(* CoDeSys 2.3.9.40 project: Атмосфера 02.12.15.pro *)
(* Libraries: Util.lib 18.5.10 14:14:28, STANDARD.LIB 4.10.05 10:14:46, IECSFC.LIB 13.4.06 14:51:28, ANALYZATION.LIB 5.10.99 08:05:06 *)

(* PLC configuration (modules and I/O channels)
Fast discrete inputs [I_SIMPLE_INPUT] node 0, in %IB0 out %QB0 {Filtrationtime = 10}
  AT %IX0.0 [BitInput] PUSK_SYS
  AT %IX0.1 [BitInput] STOP_SYS
  AT %IX0.2 [BitInput] gribok
  AT %IX0.3 [BitInput] avto_all
Discrete inputs [ID130] node 1, in %IB1 out %QB1 {Filtrationtime_GeneralINP = 10; Visibility = No; PinCount = 32}
  AT %IB1.0 [ByteInput] 8 discrete inputs
  AT %IB1.1 [ByteInput] 8 discrete inputs
  AT %IB1.2 [ByteInput] 8 discrete inputs
  AT %IB1.3 [ByteInput] 8 discrete inputs
Fast discrete outputs [OWEN_ID570] node 2, in %IB2 out %QB2 {SafeValueBool = FALSE; SafeValueBool = FALSE; SafeValueBool = FALSE; SafeValueBool = FALSE; Visibility = No}
  AT %QX2.0 [BitOutput] ready_LK3
  AT %QX2.1 [BitOutput] avaria
  AT %QX2.2 [BitOutput] metall
  AT %QX2.3 [BitOutput] ready_LK10
Discrete outputs [ID131] node 3, in %IB3 out %QB3 {SafeValueByte = 0; SafeValueByte = 0; SafeValueByteM = 0; Visibility = No; PinCount = 24}
  AT %QB3.0 [ByteOutput] 8 discrete outputs
  AT %QB3.1 [ByteOutput] 8 discrete outputs
  AT %QB3.2 [ByteOutput] 4 discrete outputs
Special input [ID103] node 4, in %IB4 out %QB4 {Filtrationtime = 1000; PinCount = 1; WatchDogPeriod = 400; PollPeriod = 3000; Visibility = No}
  AT %IX4.0 [BitInput] Special input
Special output [ID104] node 5, in %IB5 out %QB5 {Visibility = No; PinCount = 1}
  AT %QX5.0 [BitOutput] Special output
Button [ID003] node 6, in %IB6 out %QB6
  AT %IX6.0 [BitInput] Button Start/Stop
ModBus (Master) [MODBUS_MASTER_ID450] node 7, in %IB7 out %QB7 {Visibility = No}
  AT %QD7.0 [DWordOutput] Last address
  AT %QW7.1 [WordOutput] Last error
  RS-485-2 [COM3_USART] node 0, in %IB7.0 out %QB7.0 {CommunicationSpeed = 38400; Parity = NO PARITY CHECK; BitLength = 8 bits; StopLength = One stop bit; InterfaceType = RS485; FrameOriented = RTU; Timeout = 0; Visibility = No}
  Universal Modbus device [ID2000] node 1, in %IB7.1 out %QB7.1 {ModuleIP = 10:0:0:223; ServiceTimeout = 150; TCPport = 502; NetMode = Serial; ModuleSlaveAddress = 10; RequestType = By poll time; PeriodOfService = 100; Visibility = No; RepeatCounter = 0; ByteSequence = Trace_mode}
    AT %QB7.1.0 [ComChannel] LK10
AT %IB7.1.0.0 [ByteInput]
AT %QW7.1.1.0 [WordOutput] KM1_LK10
AT %IW7.1.2.0 [WordInput]
Universal Modbus device [ID2000] node 2, in %IB7.2 out %QB7.2 {ModuleIP = 10:0:0:223; ServiceTimeout = 150; TCPport = 502; NetMode = Serial; ModuleSlaveAddress = 11; RequestType = By poll time; PeriodOfService = 100; Visibility = No; RepeatCounter = 0; ByteSequence = Trace_mode}
  AT %QB7.2.0 [ComChannel] LK11
AT %IB7.2.0.0 [ByteInput]
AT %QW7.2.1.0 [WordOutput] KM1_LK11
AT %IW7.2.2.0 [WordInput]
Universal Modbus device [ID2000] node 3, in %IB7.3 out %QB7.3 {ModuleIP = 10:0:0:223; ServiceTimeout = 150; TCPport = 502; NetMode = Serial; ModuleSlaveAddress = 12; RequestType = By poll time; PeriodOfService = 100; Visibility = No; RepeatCounter = 0; ByteSequence = Trace_mode}
  AT %QB7.3.0 [ComChannel] LK12
AT %IB7.3.0.0 [ByteInput]
AT %QW7.3.1.0 [WordOutput] KM1_LK12
AT %IW7.3.2.0 [WordInput]
Universal Modbus device [ID2000] node 4, in %IB7.4 out %QB7.4 {ModuleIP = 10:0:0:223; ServiceTimeout = 150; TCPport = 502; NetMode = Serial; ModuleSlaveAddress = 13; RequestType = By poll time; PeriodOfService = 100; Visibility = No; RepeatCounter = 0; ByteSequence = Trace_mode}
  AT %QB7.4.0 [ComChannel] LK13
AT %IB7.4.0.0 [ByteInput]
AT %QW7.4.1.0 [WordOutput] KM1_LK13
AT %IW7.4.2.0 [WordInput]
Universal Modbus device [ID2000] node 5, in %IB7.5 out %QB7.5 {ModuleIP = 10:0:0:223; ServiceTimeout = 150; TCPport = 502; NetMode = Serial; ModuleSlaveAddress = 14; RequestType = By poll time; PeriodOfService = 100; Visibility = No; RepeatCounter = 0; ByteSequence = Trace_mode}
  AT %QB7.5.0 [ComChannel] GR3
AT %IB7.5.0.0 [ByteInput]
AT %QW7.5.1.0 [WordOutput] KM1_GR3
Universal Modbus device [ID2000] node 6, in %IB7.6 out %QB7.6 {ModuleIP = 10:0:0:223; ServiceTimeout = 150; TCPport = 502; NetMode = Serial; ModuleSlaveAddress = 6; RequestType = By poll time; PeriodOfService = 100; Visibility = No; RepeatCounter = 0; ByteSequence = Trace_mode}
  AT %QB7.6.0 [ComChannel] LK6
AT %IB7.6.0.0 [ByteInput]
AT %QW7.6.1.0 [WordOutput] KM1_LK6
AT %IW7.6.2.0 [WordInput]
Universal Modbus device [ID2000] node 7, in %IB7.7 out %QB7.7 {ModuleIP = 10:0:0:223; ServiceTimeout = 150; TCPport = 502; NetMode = Serial; ModuleSlaveAddress = 9; RequestType = By poll time; PeriodOfService = 100; Visibility = No; RepeatCounter = 0; ByteSequence = Trace_mode}
  AT %QB7.7.0 [ComChannel] LK9
AT %IB7.7.0.0 [ByteInput]
AT %QW7.7.1.0 [WordOutput] KM1_LK9
AT %IW7.7.2.0 [WordInput]
Universal Modbus device [ID2000] node 8, in %IB7.8 out %QB7.8 {ModuleIP = 10:0:0:223; ServiceTimeout = 150; TCPport = 502; NetMode = Serial; ModuleSlaveAddress = 18; RequestType = By poll time; PeriodOfService = 100; Visibility = No; RepeatCounter = 0; ByteSequence = Trace_mode}
  AT %QB7.8.0 [ComChannel] LP1_3 mod1
AT %IB7.8.0.0 [ByteInput]
AT %QW7.8.1.0 [WordOutput] KM1_LP1_3
Universal Modbus device [ID2000] node 9, in %IB7.9 out %QB7.9 {ModuleIP = 10:0:0:223; ServiceTimeout = 150; TCPport = 502; NetMode = Serial; ModuleSlaveAddress = 19; RequestType = By poll time; PeriodOfService = 100; Visibility = No; RepeatCounter = 0; ByteSequence = Trace_mode}
  AT %QB7.9.0 [ComChannel] LP1_3 mod2
AT %IB7.9.0.0 [ByteInput]
AT %QW7.9.1.0 [WordOutput] KM2345_LP1_3_byte
AT %IW7.9.2.0 [WordInput]
AT %IW7.9.3.0 [WordInput]
AT %IW7.9.4.0 [WordInput]
Universal Modbus device [ID2000] node 10, in %IB7.10 out %QB7.10 {ModuleIP = 10:0:0:223; ServiceTimeout = 150; TCPport = 502; NetMode = Serial; ModuleSlaveAddress = 15; RequestType = By poll time; PeriodOfService = 100; Visibility = No; RepeatCounter = 0; ByteSequence = Trace_mode}
  AT %QB7.10.0 [ComChannel] GR2
AT %IB7.10.0.0 [ByteInput]
AT %QW7.10.1.0 [WordOutput] KM1_GR2
Universal Modbus device [ID2000] node 11, in %IB7.11 out %QB7.11 {ModuleIP = 10:0:0:223; ServiceTimeout = 150; TCPport = 502; NetMode = Serial; ModuleSlaveAddress = 4; RequestType = By poll time; PeriodOfService = 100; Visibility = No; RepeatCounter = 0; ByteSequence = Trace_mode}
  AT %QB7.11.0 [ComChannel] LK4
AT %IB7.11.0.0 [ByteInput]
AT %QW7.11.1.0 [WordOutput] KM1_LK4
AT %IW7.11.2.0 [WordInput]
Universal Modbus device [ID2000] node 12, in %IB7.12 out %QB7.12 {ModuleIP = 10:0:0:223; ServiceTimeout = 150; TCPport = 502; NetMode = Serial; ModuleSlaveAddress = 1; RequestType = By poll time; PeriodOfService = 100; Visibility = No; RepeatCounter = 0; ByteSequence = Trace_mode}
  AT %QB7.12.0 [ComChannel] GR1
AT %IB7.12.0.0 [ByteInput]
AT %QW7.12.1.0 [WordOutput] KM1_GR1
Universal Modbus device [ID2000] node 13, in %IB7.13 out %QB7.13 {ModuleIP = 10:0:0:223; ServiceTimeout = 150; TCPport = 502; NetMode = Serial; ModuleSlaveAddress = 2; RequestType = By poll time; PeriodOfService = 100; Visibility = No; RepeatCounter = 0; ByteSequence = Trace_mode}
  AT %QB7.13.0 [ComChannel] LK2
AT %IB7.13.0.0 [ByteInput]
AT %QW7.13.1.0 [WordOutput] KM1_LK2
AT %IW7.13.2.0 [WordInput]
Universal Modbus device [ID2000] node 14, in %IB7.14 out %QB7.14 {ModuleIP = 10:0:0:223; ServiceTimeout = 150; TCPport = 502; NetMode = Serial; ModuleSlaveAddress = 3; RequestType = By poll time; PeriodOfService = 100; Visibility = No; RepeatCounter = 0; ByteSequence = Trace_mode}
  AT %QB7.14.0 [ComChannel] LK3
AT %IB7.14.0.0 [ByteInput]
AT %QW7.14.1.0 [WordOutput] KM1_LK3
AT %IW7.14.2.0 [WordInput]
Universal Modbus device [ID2000] node 15, in %IB7.15 out %QB7.15 {ModuleIP = 10:0:0:223; ServiceTimeout = 150; TCPport = 502; NetMode = Serial; ModuleSlaveAddress = 20; RequestType = By poll time; PeriodOfService = 100; Visibility = No; RepeatCounter = 0; ByteSequence = Trace_mode}
  AT %QB7.15.0 [ComChannel] VP1
AT %IB7.15.0.0 [ByteInput]
AT %QW7.15.1.0 [WordOutput]
Universal Modbus device [ID2000] node 16, in %IB7.16 out %QB7.16 {ModuleIP = 10:0:0:223; ServiceTimeout = 150; TCPport = 502; NetMode = Serial; ModuleSlaveAddress = 27; RequestType = By poll time; PeriodOfService = 100; Visibility = No; RepeatCounter = 0; ByteSequence = Trace_mode}
  AT %QB7.16.0 [ComChannel] Command (0xff - Start)
AT %IB7.16.0.0 [ByteInput]
AT %QW7.16.1.0 [WordOutput] km_byte_cyc
Universal Modbus device [ID2000] node 17, in %IB7.17 out %QB7.17 {ModuleIP = 10:0:0:223; ServiceTimeout = 150; TCPport = 502; NetMode = Serial; ModuleSlaveAddress = 26; RequestType = By poll time; PeriodOfService = 100; Visibility = No; RepeatCounter = 0; ByteSequence = Trace_mode}
  AT %QB7.17.0 [ComChannel] Command (0xff - Start)
AT %QW7.17.0.0 [WordOutput]
AT %QW7.17.1.0 [WordOutput]
AT %QW7.17.2.0 [WordOutput]
AT %QW7.17.3.0 [WordOutput]
AT %QW7.17.4.0 [WordOutput]
AT %QW7.17.5.0 [WordOutput]
AT %QW7.17.6.0 [WordOutput]
AT %QW7.17.7.0 [WordOutput]
Universal Modbus device [ID2000] node 18, in %IB7.18 out %QB7.18 {ModuleIP = 10:0:0:223; ServiceTimeout = 150; TCPport = 502; NetMode = Serial; ModuleSlaveAddress = 44; RequestType = By poll time; PeriodOfService = 100; Visibility = No; RepeatCounter = 0; ByteSequence = Trace_mode}
  AT %QB7.18.0 [ComChannel] Command (0xff - Start)
AT %ID7.18.0.0 [FloatInput]
AT %ID7.18.1.0 [FloatInput]
ModBus (slave) [MODBUS_ID400] node 8, in %IB8 out %QB8 {SlaveIdentificator = 1; Visibility = No}
  Modbus [MODBUS_ID302] node 0, in %IB8.0 out %QB8.0
    TCP [TCP_ID221] node 0, in %IB8.0.0 out %QB8.0.0 {RemotePort = 502; Visibility = No}
  8 bits [8Bit] node 1, in %IB8.1 out %QB8.1
    AT %QB8.1.0 [ByteOutput]
  8 bits [8Bit] node 2, in %IB8.2 out %QB8.2
    AT %QB8.2.0 [ByteOutput]
  8 bits [8Bit] node 3, in %IB8.3 out %QB8.3
    AT %QB8.3.0 [ByteOutput]
  8 bits [8Bit] node 4, in %IB8.4 out %QB8.4
    AT %QB8.4.0 [ByteOutput]
  8 bits [8Bit] node 5, in %IB8.5 out %QB8.5
    AT %QB8.5.0 [ByteOutput]
  8 bits [8Bit] node 6, in %IB8.6 out %QB8.6
    AT %QB8.6.0 [ByteOutput]
  8 bits [8Bit] node 7, in %IB8.7 out %QB8.7
    AT %QB8.7.0 [ByteOutput]
  8 bits [8Bit] node 8, in %IB8.8 out %QB8.8
    AT %QB8.8.0 [ByteOutput]
  8 bits [8Bit] node 9, in %IB8.9 out %QB8.9
    AT %QB8.9.0 [ByteOutput]
  8 bits [8Bit] node 10, in %IB8.10 out %QB8.10
    AT %QB8.10.0 [ByteOutput]
  8 bits [8Bit] node 11, in %IB8.11 out %QB8.11
    AT %QB8.11.0 [ByteOutput]
  8 bits [8Bit] node 12, in %IB8.12 out %QB8.12
    AT %QB8.12.0 [ByteOutput]
  8 bits [8Bit] node 13, in %IB8.13 out %QB8.13
    AT %QB8.13.0 [ByteOutput]
  8 bits [8Bit] node 14, in %IB8.14 out %QB8.14
    AT %QB8.14.0 [ByteOutput]
  8 bits [8Bit] node 15, in %IB8.15 out %QB8.15
    AT %QB8.15.0 [ByteOutput]
  8 bits [8Bit] node 16, in %IB8.16 out %QB8.16
    AT %QB8.16.0 [ByteOutput]
  8 bits [8Bit] node 17, in %IB8.17 out %QB8.17
    AT %QB8.17.0 [ByteOutput]
  8 bits [8Bit] node 18, in %IB8.18 out %QB8.18
    AT %QB8.18.0 [ByteOutput]
  8 bits [8Bit] node 19, in %IB8.19 out %QB8.19
    AT %QB8.19.0 [ByteOutput]
  8 bits [8Bit] node 20, in %IB8.20 out %QB8.20
    AT %QB8.20.0 [ByteOutput]
  8 bits [8Bit] node 21, in %IB8.21 out %QB8.21
    AT %QB8.21.0 [ByteOutput]
  8 bits [8Bit] node 22, in %IB8.22 out %QB8.22
    AT %QB8.22.0 [ByteOutput]
  8 bits [8Bit] node 23, in %IB8.23 out %QB8.23
    AT %QB8.23.0 [ByteOutput]
  8 bits [8Bit] node 24, in %IB8.24 out %QB8.24
    AT %QB8.24.0 [ByteOutput]
  8 bits [8Bit] node 25, in %IB8.25 out %QB8.25
    AT %QB8.25.0 [ByteOutput]
  8 bits [8Bit] node 26, in %IB8.26 out %QB8.26
    AT %QB8.26.0 [ByteOutput]
  8 bits [8Bit] node 27, in %IB8.27 out %QB8.27
    AT %QB8.27.0 [ByteOutput]
  8 bits [8Bit] node 28, in %IB8.28 out %QB8.28
    AT %QB8.28.0 [ByteOutput]
  8 bits [8Bit] node 29, in %IB8.29 out %QB8.29
    AT %QB8.29.0 [ByteOutput]
  8 bits [8Bit] node 30, in %IB8.30 out %QB8.30
    AT %QB8.30.0 [ByteOutput]
  8 bits [8Bit] node 31, in %IB8.31 out %QB8.31
    AT %QB8.31.0 [ByteOutput]
  2 byte [Register] node 32, in %IB8.32 out %QB8.32
    AT %QW8.32.0 [WordOutput] input_Hz_LP4
  2 byte [Register] node 33, in %IB8.33 out %QB8.33
    AT %QW8.33.0 [WordOutput] input_Hz_LP5
  2 byte [Register] node 34, in %IB8.34 out %QB8.34
    AT %QW8.34.0 [WordOutput] LV_GR1_out
  2 byte [Register] node 35, in %IB8.35 out %QB8.35
    AT %QW8.35.0 [WordOutput] LV_LK7_out
  2 byte [Register] node 36, in %IB8.36 out %QB8.36
    AT %QW8.36.0 [WordOutput] LV_LK8_out
  2 byte [Register] node 37, in %IB8.37 out %QB8.37
    AT %QW8.37.0 [WordOutput] output_Hz_LP4_out
  2 byte [Register] node 38, in %IB8.38 out %QB8.38
    AT %QW8.38.0 [WordOutput] output_Hz_LP5_out
  2 byte [Register] node 39, in %IB8.39 out %QB8.39
    AT %QW8.39.0 [WordOutput] LV_D2_out
  Float [Float] node 40, in %IB8.40 out %QB8.40
    AT %QD8.40.0 [FloatOutput] ust_LV2_GR1
  Float [Float] node 41, in %IB8.41 out %QB8.41
    AT %QD8.41.0 [FloatOutput] ust_LV1_GR1
  Float [Float] node 42, in %IB8.42 out %QB8.42
    AT %QD8.42.0 [FloatOutput] ust_LV2_LK7
  Float [Float] node 43, in %IB8.43 out %QB8.43
    AT %QD8.43.0 [FloatOutput] ust_LV1_LK7
  Float [Float] node 44, in %IB8.44 out %QB8.44
    AT %QD8.44.0 [FloatOutput] ust_LV1_LK7
  Float [Float] node 45, in %IB8.45 out %QB8.45
    AT %QD8.45.0 [FloatOutput] ust_LV1_LK7
  Float [Float] node 46, in %IB8.46 out %QB8.46
    AT %QD8.46.0 [FloatOutput] ust_LV1_LK7
  Float [Float] node 47, in %IB8.47 out %QB8.47
    AT %QD8.47.0 [FloatOutput] ust_LV1_LK7
  2 byte [Register] node 48, in %IB8.48 out %QB8.48
    AT %QW8.48.0 [WordOutput] pusk_LAN_LP4
  2 byte [Register] node 49, in %IB8.49 out %QB8.49
    AT %QW8.49.0 [WordOutput] stop_LAN_LP4
  2 byte [Register] node 50, in %IB8.50 out %QB8.50
    AT %QW8.50.0 [WordOutput] pusk_LAN_LP5
  2 byte [Register] node 51, in %IB8.51 out %QB8.51
    AT %QW8.51.0 [WordOutput] stop_LAN_LP5
  2 byte [Register] node 52, in %IB8.52 out %QB8.52
    AT %QW8.52.0 [WordOutput] pusk_LAN_VP1
  2 byte [Register] node 53, in %IB8.53 out %QB8.53
    AT %QW8.53.0 [WordOutput] stop_LAN_VP1
  2 byte [Register] node 54, in %IB8.54 out %QB8.54
    AT %QW8.54.0 [WordOutput] pusk_lan_LK10
  2 byte [Register] node 55, in %IB8.55 out %QB8.55
    AT %QW8.55.0 [WordOutput] pusk_lan_LK11
  2 byte [Register] node 56, in %IB8.56 out %QB8.56
    AT %QW8.56.0 [WordOutput] pusk_lan_LK12
  2 byte [Register] node 57, in %IB8.57 out %QB8.57
    AT %QW8.57.0 [WordOutput] pusk_lan_LK13
  2 byte [Register] node 58, in %IB8.58 out %QB8.58
    AT %QW8.58.0 [WordOutput] pusk_lan_GR3
  2 byte [Register] node 59, in %IB8.59 out %QB8.59
    AT %QW8.59.0 [WordOutput] pusk_lan_LK7
  2 byte [Register] node 60, in %IB8.60 out %QB8.60
    AT %QW8.60.0 [WordOutput] pusk_lan_LK8
  2 byte [Register] node 61, in %IB8.61 out %QB8.61
    AT %QW8.61.0 [WordOutput] pusk_lan_LK6
  2 byte [Register] node 62, in %IB8.62 out %QB8.62
    AT %QW8.62.0 [WordOutput] pusk_lan_LK9
  2 byte [Register] node 63, in %IB8.63 out %QB8.63
    AT %QW8.63.0 [WordOutput] pusk_lan_LP1_3
  2 byte [Register] node 64, in %IB8.64 out %QB8.64
    AT %QW8.64.0 [WordOutput] pusk_lan_GR2
  2 byte [Register] node 65, in %IB8.65 out %QB8.65
    AT %QW8.65.0 [WordOutput] pusk_lan_LK5
  2 byte [Register] node 66, in %IB8.66 out %QB8.66
    AT %QW8.66.0 [WordOutput] pusk_lan_LK4
  2 byte [Register] node 67, in %IB8.67 out %QB8.67
    AT %QW8.67.0 [WordOutput] pusk_lan_LK3
  2 byte [Register] node 68, in %IB8.68 out %QB8.68
    AT %QW8.68.0 [WordOutput] pusk_lan_GR1
  2 byte [Register] node 69, in %IB8.69 out %QB8.69
    AT %QW8.69.0 [WordOutput] pusk_lan_LK2
  2 byte [Register] node 70, in %IB8.70 out %QB8.70
    AT %QW8.70.0 [WordOutput] stop_lan_LK10
  2 byte [Register] node 71, in %IB8.71 out %QB8.71
    AT %QW8.71.0 [WordOutput] stop_lan_LK11
  2 byte [Register] node 72, in %IB8.72 out %QB8.72
    AT %QW8.72.0 [WordOutput] stop_lan_LK12
  2 byte [Register] node 73, in %IB8.73 out %QB8.73
    AT %QW8.73.0 [WordOutput] stop_lan_LK13
  2 byte [Register] node 74, in %IB8.74 out %QB8.74
    AT %QW8.74.0 [WordOutput] stop_lan_GR3
  2 byte [Register] node 75, in %IB8.75 out %QB8.75
    AT %QW8.75.0 [WordOutput] stop_lan_LK7
  2 byte [Register] node 76, in %IB8.76 out %QB8.76
    AT %QW8.76.0 [WordOutput] stop_lan_LK8
  2 byte [Register] node 77, in %IB8.77 out %QB8.77
    AT %QW8.77.0 [WordOutput] stop_lan_LK6
  2 byte [Register] node 78, in %IB8.78 out %QB8.78
    AT %QW8.78.0 [WordOutput] stop_lan_LK9
  2 byte [Register] node 79, in %IB8.79 out %QB8.79
    AT %QW8.79.0 [WordOutput] stop_lan_LP1_3
  2 byte [Register] node 80, in %IB8.80 out %QB8.80
    AT %QW8.80.0 [WordOutput] stop_lan_GR2
  2 byte [Register] node 81, in %IB8.81 out %QB8.81
    AT %QW8.81.0 [WordOutput] stop_lan_LK5
  2 byte [Register] node 82, in %IB8.82 out %QB8.82
    AT %QW8.82.0 [WordOutput] stop_lan_LK4
  2 byte [Register] node 83, in %IB8.83 out %QB8.83
    AT %QW8.83.0 [WordOutput] stop_lan_LK3
  2 byte [Register] node 84, in %IB8.84 out %QB8.84
    AT %QW8.84.0 [WordOutput] stop_lan_GR1
  2 byte [Register] node 85, in %IB8.85 out %QB8.85
    AT %QW8.85.0 [WordOutput] stop_lan_LK2
  2 byte [Register] node 86, in %IB8.86 out %QB8.86
    AT %QW8.86.0 [WordOutput] stop_LAN_D3
  2 byte [Register] node 87, in %IB8.87 out %QB8.87
    AT %QW8.87.0 [WordOutput] stop_LAN_D4
  2 byte [Register] node 88, in %IB8.88 out %QB8.88
    AT %QW8.88.0 [WordOutput] stop_LAN_D2
  2 byte [Register] node 89, in %IB8.89 out %QB8.89
    AT %QW8.89.0 [WordOutput] pusk_LAN_D2
  2 byte [Register] node 90, in %IB8.90 out %QB8.90
    AT %QW8.90.0 [WordOutput] pusk_LAN_D3
  2 byte [Register] node 91, in %IB8.91 out %QB8.91
    AT %QW8.91.0 [WordOutput] pusk_LAN_D4
  2 byte [Register] node 92, in %IB8.92 out %QB8.92
    AT %QW8.92.0 [WordOutput] pusk_lan_cyclone
  2 byte [Register] node 93, in %IB8.93 out %QB8.93
    AT %QW8.93.0 [WordOutput] stop_lan_cyclone
  Float [Float] node 94, in %IB8.94 out %QB8.94
    AT %QD8.94.0 [FloatOutput] skvaj_in
  Float [Float] node 95, in %IB8.95 out %QB8.95
    AT %QD8.95.0 [FloatOutput] skvaj1_in
  Float [Float] node 96, in %IB8.96 out %QB8.96
    AT %QD8.96.0 [FloatOutput] skvaj2_in
  Float [Float] node 97, in %IB8.97 out %QB8.97
    AT %QD8.97.0 [FloatOutput] skvaj3_in
  Float [Float] node 98, in %IB8.98 out %QB8.98
    AT %QD8.98.0 [FloatOutput] skvaj4_in
  Float [Float] node 99, in %IB8.99 out %QB8.99
    AT %QD8.99.0 [FloatOutput] skvaj5_in
  Float [Float] node 100, in %IB8.100 out %QB8.100
    AT %QD8.100.0 [FloatOutput] skvaj6_in
  Float [Float] node 101, in %IB8.101 out %QB8.101
    AT %QD8.101.0 [FloatOutput] skvaj7_in
  2 byte [Register] node 102, in %IB8.102 out %QB8.102
    AT %QW8.102.0 [WordOutput] tros_self_lk10
  2 byte [Register] node 103, in %IB8.103 out %QB8.103
    AT %QW8.103.0 [WordOutput] shod_self_lk10
  2 byte [Register] node 104, in %IB8.104 out %QB8.104
    AT %QW8.104.0 [WordOutput] ogr_self_lk10
  2 byte [Register] node 105, in %IB8.105 out %QB8.105
    AT %QW8.105.0 [WordOutput] vl_self_lk10
  2 byte [Register] node 106, in %IB8.106 out %QB8.106
    AT %QW8.106.0 [WordOutput] tros_self_lk11
  2 byte [Register] node 107, in %IB8.107 out %QB8.107
    AT %QW8.107.0 [WordOutput] shod_self_lk11
  2 byte [Register] node 108, in %IB8.108 out %QB8.108
    AT %QW8.108.0 [WordOutput] ogr_self_lk11
  2 byte [Register] node 109, in %IB8.109 out %QB8.109
    AT %QW8.109.0 [WordOutput] vl_self_lk11
  2 byte [Register] node 110, in %IB8.110 out %QB8.110
    AT %QW8.110.0 [WordOutput] tros_self_lk12
  2 byte [Register] node 111, in %IB8.111 out %QB8.111
    AT %QW8.111.0 [WordOutput] shod_self_lk12
  2 byte [Register] node 112, in %IB8.112 out %QB8.112
    AT %QW8.112.0 [WordOutput] ogr_self_lk12
  2 byte [Register] node 113, in %IB8.113 out %QB8.113
    AT %QW8.113.0 [WordOutput] vl_self_lk12
  2 byte [Register] node 114, in %IB8.114 out %QB8.114
    AT %QW8.114.0 [WordOutput] tros_self_lk13
  2 byte [Register] node 115, in %IB8.115 out %QB8.115
    AT %QW8.115.0 [WordOutput] shod_self_lk13
  2 byte [Register] node 116, in %IB8.116 out %QB8.116
    AT %QW8.116.0 [WordOutput] ogr_self_lk13
  2 byte [Register] node 117, in %IB8.117 out %QB8.117
    AT %QW8.117.0 [WordOutput] vl_self_lk13
  2 byte [Register] node 118, in %IB8.118 out %QB8.118
    AT %QW8.118.0 [WordOutput] tros_self_lk7
  2 byte [Register] node 119, in %IB8.119 out %QB8.119
    AT %QW8.119.0 [WordOutput] shod_self_lk7
  2 byte [Register] node 120, in %IB8.120 out %QB8.120
    AT %QW8.120.0 [WordOutput] ogr_self_lk7
  2 byte [Register] node 121, in %IB8.121 out %QB8.121
    AT %QW8.121.0 [WordOutput] vl_self_lk7
  2 byte [Register] node 122, in %IB8.122 out %QB8.122
    AT %QW8.122.0 [WordOutput] ogr_self_lk7
  2 byte [Register] node 123, in %IB8.123 out %QB8.123
    AT %QW8.123.0 [WordOutput] shod_self_lk8
  2 byte [Register] node 124, in %IB8.124 out %QB8.124
    AT %QW8.124.0 [WordOutput] ogr_self_lk8
  2 byte [Register] node 125, in %IB8.125 out %QB8.125
    AT %QW8.125.0 [WordOutput] vl_self_lk8
  2 byte [Register] node 126, in %IB8.126 out %QB8.126
    AT %QW8.126.0 [WordOutput] tros_self_lk6
  2 byte [Register] node 127, in %IB8.127 out %QB8.127
    AT %QW8.127.0 [WordOutput] shod_self_lk6
  2 byte [Register] node 128, in %IB8.128 out %QB8.128
    AT %QW8.128.0 [WordOutput] ogr_self_lk6
  2 byte [Register] node 129, in %IB8.129 out %QB8.129
    AT %QW8.129.0 [WordOutput] vl_self_lk6
  2 byte [Register] node 130, in %IB8.130 out %QB8.130
    AT %QW8.130.0 [WordOutput] tros_self_lk9
  2 byte [Register] node 131, in %IB8.131 out %QB8.131
    AT %QW8.131.0 [WordOutput] shod_self_lk9
  2 byte [Register] node 132, in %IB8.132 out %QB8.132
    AT %QW8.132.0 [WordOutput] ogr_self_lk9
  2 byte [Register] node 133, in %IB8.133 out %QB8.133
    AT %QW8.133.0 [WordOutput] vl_self_lk9
  2 byte [Register] node 134, in %IB8.134 out %QB8.134
    AT %QW8.134.0 [WordOutput] vl_self_lp1_3
  2 byte [Register] node 135, in %IB8.135 out %QB8.135
    AT %QW8.135.0 [WordOutput] tros_self_lk5
  2 byte [Register] node 136, in %IB8.136 out %QB8.136
    AT %QW8.136.0 [WordOutput] shod_self_lk5
  2 byte [Register] node 137, in %IB8.137 out %QB8.137
    AT %QW8.137.0 [WordOutput] ogr_self_lk5
  2 byte [Register] node 138, in %IB8.138 out %QB8.138
    AT %QW8.138.0 [WordOutput] vl_self_lk5
  2 byte [Register] node 139, in %IB8.139 out %QB8.139
    AT %QW8.139.0 [WordOutput] tros_self_lk4
  2 byte [Register] node 140, in %IB8.140 out %QB8.140
    AT %QW8.140.0 [WordOutput] shod_self_lk4
  2 byte [Register] node 141, in %IB8.141 out %QB8.141
    AT %QW8.141.0 [WordOutput] vl_self_lk4
  2 byte [Register] node 142, in %IB8.142 out %QB8.142
    AT %QW8.142.0 [WordOutput] tros_self_lk3
  2 byte [Register] node 143, in %IB8.143 out %QB8.143
    AT %QW8.143.0 [WordOutput] shod_self_lk3
  2 byte [Register] node 144, in %IB8.144 out %QB8.144
    AT %QW8.144.0 [WordOutput] ogr_self_lk3
  2 byte [Register] node 145, in %IB8.145 out %QB8.145
    AT %QW8.145.0 [WordOutput] vl_self_lk3
  2 byte [Register] node 146, in %IB8.146 out %QB8.146
    AT %QW8.146.0 [WordOutput] vl_self_lk3
  2 byte [Register] node 147, in %IB8.147 out %QB8.147
    AT %QW8.147.0 [WordOutput] shod_self_lk2
  2 byte [Register] node 148, in %IB8.148 out %QB8.148
    AT %QW8.148.0 [WordOutput] ogr_self_lk2
  2 byte [Register] node 149, in %IB8.149 out %QB8.149
    AT %QW8.149.0 [WordOutput] vl_self_lk2
  2 byte [Register] node 150, in %IB8.150 out %QB8.150
    AT %QW8.150.0 [WordOutput] revers
  2 byte [Register] node 151, in %IB8.151 out %QB8.151
    AT %QW8.151.0 [WordOutput] vl_self_lp4
  2 byte [Register] node 152, in %IB8.152 out %QB8.152
    AT %QW8.152.0 [WordOutput] vl_self_lp5
  8 bits [8Bit] node 153, in %IB8.153 out %QB8.153
    AT %QB8.153.0 [ByteOutput]
  8 bits [8Bit] node 154, in %IB8.154 out %QB8.154
    AT %QB8.154.0 [ByteOutput]
  2 byte [Register] node 155, in %IB8.155 out %QB8.155
    AT %QW8.155.0 [WordOutput]
  2 byte [Register] node 156, in %IB8.156 out %QB8.156
    AT %QW8.156.0 [WordOutput]
  2 byte [Register] node 157, in %IB8.157 out %QB8.157
    AT %QW8.157.0 [WordOutput]
  2 byte [Register] node 158, in %IB8.158 out %QB8.158
    AT %QW8.158.0 [WordOutput]
  8 bits [8Bit] node 159, in %IB8.159 out %QB8.159
    AT %QB8.159.0 [ByteOutput]
  2 byte [Register] node 160, in %IB8.160 out %QB8.160
    AT %QW8.160.0 [WordOutput]
  2 byte [Register] node 161, in %IB8.161 out %QB8.161
    AT %QW8.161.0 [WordOutput]
  2 byte [Register] node 162, in %IB8.162 out %QB8.162
    AT %QW8.162.0 [WordOutput]
  2 byte [Register] node 163, in %IB8.163 out %QB8.163
    AT %QW8.163.0 [WordOutput]
  2 byte [Register] node 164, in %IB8.164 out %QB8.164
    AT %QW8.164.0 [WordOutput]
  2 byte [Register] node 165, in %IB8.165 out %QB8.165
    AT %QW8.165.0 [WordOutput]
  2 byte [Register] node 166, in %IB8.166 out %QB8.166
    AT %QW8.166.0 [WordOutput]
  8 bits [8Bit] node 167, in %IB8.167 out %QB8.167
    AT %QB8.167.0 [ByteOutput]
AT %QW8.168.0 [WordOutput]
AT %QD9.0 [DWordOutput] Last address
AT %QW9.1 [WordOutput] Last error
RS-485-1 [COM1_USART] node 0, in %IB9.0 out %QB9.0 {CommunicationSpeed = 38400; Parity = NO PARITY CHECK; BitLength = 8 bits; StopLength = One stop bit; InterfaceType = RS485; FrameOriented = RTU; Timeout = 0; Visibility = No}
Universal Modbus device [ID2000] node 1, in %IB9.1 out %QB9.1 {ModuleIP = 10:0:0:223; ServiceTimeout = 150; TCPport = 502; NetMode = Serial; ModuleSlaveAddress = 3; RequestType = By poll time; PeriodOfService = 100; Visibility = No; RepeatCounter = 0; ByteSequence = Trace_mode}
  AT %QB9.1.0 [ComChannel] Command (0xff - Start)
AT %IW9.1.0.0 [WordInput]
Universal Modbus device [ID2000] node 2, in %IB9.2 out %QB9.2 {ModuleIP = 10:0:0:223; ServiceTimeout = 150; TCPport = 502; NetMode = Serial; ModuleSlaveAddress = 2; RequestType = By poll time; PeriodOfService = 100; Visibility = No; RepeatCounter = 0; ByteSequence = Trace_mode}
  AT %QB9.2.0 [ComChannel] Command (0xff - Start)
AT %IW9.2.0.0 [WordInput]
Universal Modbus device [ID2000] node 3, in %IB9.3 out %QB9.3 {ModuleIP = 10:0:0:223; ServiceTimeout = 150; TCPport = 502; NetMode = Serial; ModuleSlaveAddress = 1; RequestType = By poll time; PeriodOfService = 100; Visibility = No; RepeatCounter = 0; ByteSequence = Trace_mode}
  AT %QB9.3.0 [ComChannel] Command (0xff - Start)
AT %ID9.3.0.0 [FloatInput]
AT %ID9.3.1.0 [FloatInput]
Universal Modbus device [ID2000] node 4, in %IB9.4 out %QB9.4 {ModuleIP = 10:0:0:223; ServiceTimeout = 150; TCPport = 502; NetMode = Serial; ModuleSlaveAddress = 31; RequestType = By poll time; PeriodOfService = 100; Visibility = No; RepeatCounter = 0; ByteSequence = Trace_mode}
  AT %QB9.4.0 [ComChannel] ПЧ5
AT %QW9.4.0.0 [WordOutput] Пуск/стоп ПЧ
AT %QW9.4.1.0 [WordOutput] Изменение параметра b1.00
AT %QW9.4.2.0 [WordOutput] Изменение параметра b1.04
AT %IW9.4.3.0 [WordInput] Значение выходной частоты
AT %IW9.4.4.0 [WordInput]
Universal Modbus device [ID2000] node 5, in %IB9.5 out %QB9.5 {ModuleIP = 10:0:0:223; ServiceTimeout = 150; TCPport = 502; NetMode = Serial; ModuleSlaveAddress = 7; RequestType = By poll time; PeriodOfService = 100; Visibility = No; RepeatCounter = 0; ByteSequence = Trace_mode}
  AT %QB9.5.0 [ComChannel] LK7
AT %IB9.5.0.0 [ByteInput]
AT %QW9.5.1.0 [WordOutput] KM1_LK7
AT %IW9.5.2.0 [WordInput]
Universal Modbus device [ID2000] node 6, in %IB9.6 out %QB9.6 {ModuleIP = 10:0:0:223; ServiceTimeout = 150; TCPport = 502; NetMode = Serial; ModuleSlaveAddress = 8; RequestType = By poll time; PeriodOfService = 100; Visibility = No; RepeatCounter = 0; ByteSequence = Trace_mode}
  AT %QB9.6.0 [ComChannel] LK8
AT %IB9.6.0.0 [ByteInput]
AT %QW9.6.1.0 [WordOutput] KM1_LK8
AT %IW9.6.2.0 [WordInput]
Universal Modbus device [ID2000] node 7, in %IB9.7 out %QB9.7 {ModuleIP = 10:0:0:223; ServiceTimeout = 150; TCPport = 502; NetMode = Serial; ModuleSlaveAddress = 5; RequestType = By poll time; PeriodOfService = 100; Visibility = No; RepeatCounter = 0; ByteSequence = Trace_mode}
  AT %QB9.7.0 [ComChannel] LK5
AT %IB9.7.0.0 [ByteInput]
AT %QW9.7.1.0 [WordOutput] KM1_LK5
AT %IW9.7.2.0 [WordInput]
Universal Modbus device [ID2000] node 8, in %IB9.8 out %QB9.8 {ModuleIP = 10:0:0:223; ServiceTimeout = 150; TCPport = 502; NetMode = Serial; ModuleSlaveAddress = 16; RequestType = By poll time; PeriodOfService = 100; Visibility = No; RepeatCounter = 0; ByteSequence = Trace_mode}
  AT %QB9.8.0 [ComChannel] LP4
AT %IB9.8.0.0 [ByteInput]
AT %QW9.8.1.0 [WordOutput]
Universal Modbus device [ID2000] node 9, in %IB9.9 out %QB9.9 {ModuleIP = 10:0:0:223; ServiceTimeout = 150; TCPport = 502; NetMode = Serial; ModuleSlaveAddress = 17; RequestType = By poll time; PeriodOfService = 100; Visibility = No; RepeatCounter = 0; ByteSequence = Trace_mode}
  AT %QB9.9.0 [ComChannel] LP5
AT %IB9.9.0.0 [ByteInput]
AT %QW9.9.1.0 [WordOutput]
Universal Modbus device [ID2000] node 10, in %IB9.10 out %QB9.10 {ModuleIP = 10:0:0:223; ServiceTimeout = 150; TCPport = 502; NetMode = Serial; ModuleSlaveAddress = 24; RequestType = By poll time; PeriodOfService = 100; Visibility = No; RepeatCounter = 0; ByteSequence = Trace_mode}
  AT %QB9.10.0 [ComChannel] D3 mod1
AT %IB9.10.0.0 [ByteInput]
AT %QW9.10.1.0 [WordOutput]
AT %IW9.10.2.0 [WordInput]
Universal Modbus device [ID2000] node 11, in %IB9.11 out %QB9.11 {ModuleIP = 10:0:0:223; ServiceTimeout = 150; TCPport = 502; NetMode = Serial; ModuleSlaveAddress = 23; RequestType = By poll time; PeriodOfService = 100; Visibility = No; RepeatCounter = 0; ByteSequence = Trace_mode}
  AT %QB9.11.0 [ComChannel] D3 mod2
AT %IB9.11.0.0 [ByteInput]
Register output module [ID2004] node 1, in %IB9.11.1 out %QB9.11.1 {ModbusAddress = 50; Command_write_one_reg = Write multiple registers(0x10); Visibility = No}
  AT %QW9.11.1.0 [WordOutput]
Universal Modbus device [ID2000] node 12, in %IB9.12 out %QB9.12 {ModuleIP = 10:0:0:223; ServiceTimeout = 150; TCPport = 502; NetMode = Serial; ModuleSlaveAddress = 21; RequestType = By poll time; PeriodOfService = 100; Visibility = No; RepeatCounter = 0; ByteSequence = Trace_mode}
  AT %QB9.12.0 [ComChannel] D4 mod1
AT %IB9.12.0.0 [ByteInput]
AT %QW9.12.1.0 [WordOutput]
AT %IW9.12.2.0 [WordInput]
Universal Modbus device [ID2000] node 13, in %IB9.13 out %QB9.13 {ModuleIP = 10:0:0:223; ServiceTimeout = 150; TCPport = 502; NetMode = Serial; ModuleSlaveAddress = 22; RequestType = By poll time; PeriodOfService = 100; Visibility = No; RepeatCounter = 0; ByteSequence = Trace_mode}
  AT %QB9.13.0 [ComChannel] D4 mod2
AT %IB9.13.0.0 [ByteInput]
AT %QW9.13.1.0 [WordOutput]
Universal Modbus device [ID2000] node 14, in %IB9.14 out %QB9.14 {ModuleIP = 10:0:0:223; ServiceTimeout = 150; TCPport = 502; NetMode = Serial; ModuleSlaveAddress = 25; RequestType = By poll time; PeriodOfService = 100; Visibility = No; RepeatCounter = 0; ByteSequence = Trace_mode}
  AT %QB9.14.0 [ComChannel] D2
AT %IB9.14.0.0 [ByteInput]
AT %QW9.14.1.0 [WordOutput] KM_D2_byte
*)

(* POU PLC_PRG, LD *)
PROGRAM PLC_PRG
VAR
(*Пуск всей сисетмы в атоматическом режиме*)
	PUSK_SYS AT %IX0.0: BOOL; (*Общий пуск системы*)
	STOP_SYS AT %IX0.1: BOOL; (*По нажатию кнопки "стоп" останавливается ВП1 и ПП1*)
	prom1: BOOL; (*Самоподхват пуска уровень1*)
	prom2: BOOL; (*Самоподхват пуска уровень2*)
	prom3: BOOL; (*Самоподхват пуска уровень3*)
	prom4: BOOL; (*Самоподхват пуска уровень4*)
	prom5: BOOL; (*Самоподхват пуска уровень5*)
	prom6: BOOL; (*Самоподхват пуска уровень6*)
	prom7: BOOL; (*Самоподхват пуска уровень7*)
	prom8: BOOL; (*Самоподхват пуска уровень8*)
	prom9: BOOL; (*Самоподхват пуска уровень9*)
	avto_all AT %IX0.3:BOOL;(*Переключатель в режим автомат на шкафу контроллера*)
	gribok  AT %IX0.2:BOOL; (*Экстренна остановка завода*)
	avaria AT %QX2.1:BOOL; (*авария одного или нескольких шкафов*)
	metall AT %QX2.2:BOOL; (*Срабатывание металлдетектора*)
	pusk: BOOL; (*самоподхват пуска*)
	pusk_lan: BOOL; (*Фиксация пуска для SCADA-системы*)
	stop: CTU; (*Счетчик нажатий кнопки "стоп": после 2го нажатия останавливаются все агрегаты, кроме дробилок*)
	stop_all: BOOL; (*Подхват второго нажатия кнопки "стоп"*)
	stop_Drob: CTU; (*Счетчик нажатий кнопки "стоп": после 3го нажатия останавливаются дробилки*)
	stop_D2: BOOL; (*Подхват третьего нажатия кнопки "стоп"*)
	stop_D3: BOOL; (*Команда от дробилки Д2 на остановку дробилки Д3*)
	stop_D4: BOOL; (*Команда от дробилки Д3 на остановку дробилки Д4*)
	stop_DDD: BOOL; (*Команда от дробилки Д4 на сброс счетиков нажатий кнопки "стоп"*)
	ruchnoe_all AT %IX1.0.0:BOOL; (*Перевод завода в ручной режим: разрешение на пус отдельных агрегатов из SCADA-системы*)

(*Блок управления установуой циклона*)
	cyclone: cyclone;
	lev_up_cyc AT %IX7.16.0.0.3: BOOL; (*датчик верхнего уровня бункера*)
	lev_down_cyc AT %IX7.16.0.0.7: BOOL; (*датчик верхнего уровня бункера*)
	pre_cyc AT %IX7.16.0.0.2: BOOL; (*датчик давления*)
	ku_cyc AT %IX7.16.0.0.0: BOOL; (*контроль напряжения*)
	tz_cyc AT %IX7.16.0.0.1: BOOL; (*тепловая защита*)
	(*p_cyclone AT %IX7.16.0.0.4: BOOL; (*идикация замыкания контакторов в шкафу*)*)

	vent_pump_cyc: BOOL; (*влючение вентилятора*)
	shnek_razg AT %QX8.167.0.0: BOOL;
	shnek_up_cyc: BOOL; (*включение подъемного шнека*)
	ve1_out AT %QW7.17.0.0: WORD; (*установка скважности выхода №1*)
	ve2_out AT %QW7.17.1.0: WORD; (*установка скважности выхода №2*)
	ve3_out AT %QW7.17.2.0: WORD; (*установка скважности выхода №3*)
	ve4_out AT %QW7.17.3.0: WORD; (*установка скважности выхода №4*)
	ve5_out AT %QW7.17.4.0: WORD; (*установка скважности выхода №5*)
	ve6_out AT %QW7.17.5.0: WORD; (*установка скважности выхода №6*)
	ve7_out AT %QW7.17.6.0: WORD; (*установка скважности выхода №7*)
	ve8_out AT %QW7.17.7.0: WORD; (*установка скважности выхода №8*)
	ready_cyc: BOOL; (*готовность шкафа к работе*)
	work_cyc: BOOL; (*работа шкафа - есть давления и сумма работ контакторов*)
	avar_cyc: BOOL; (*авария шкафа*)
	km_byte_cyc AT %QW7.16.1.0: BYTE;

	(*Дробилка Д2*)
	D2: D2;
	KU_D2 AT %IX9.14.0.0.0: BOOL; (*Контроль напряжения*)
	RMS2_2 AT %IX9.14.0.0.1: BOOL; (*Работа маслостанции*)
	RD2_D2 AT %IX9.14.0.0.2: BOOL; (*Контроль работы дробилки*)
	TZD2 AT %IX9.14.0.0.3:BOOL; (*Тепловая защита дробилки Д2*)
	avto_D2 AT %IX9.14.0.0.5: BOOL; (*Выбор режима "автомат"*)
	KM_D2_byte AT %QW9.14.1.0 :BYTE; (*Битовая маска управления модулем вх/вых дробилки Д2*)

	ready_D2 AT %QX3.1.5: BOOL; (*Готовность шкафа*)
	KM2_D2: BOOL;  (*Включение контактора на звезду*)
	KM3_D2: BOOL;  (*Включение контактора на треугольник*)
	work_D2: BOOL; (*Команда разрешающая запуск следующей ступени*)

	(*Дробилка Д3*)
	D3: D3;
	KU_D3 AT %IX9.10.0.0.0: BOOL; (*Контроль напряжения шкафа управления*)
	TZN_D3 AT %IX9.10.0.0.1: BOOL; (*Тепловая защита насоса*)
	UM_D3 AT %IX9.10.0.0.2: BOOL; (*Уровень масла в маслостанции*)
	KPM_D3 AT %IX9.10.0.0.4: BOOL; (*Контроль протока масла*)
	TZV_D3 AT %IX9.10.0.0.5: BOOL; (*Тепловая защита вентилятора*)
	RMS_D3 AT %IX9.10.0.0.7: BOOL; (*Контроль работы насоса*)
	D3_mod1_byte AT %QW9.10.1.0: BYTE; (*Битовая маска управления первым модулем вх/вых дробилки Д3*)

	KUD3_D3 AT %IX9.11.0.0.0: BOOL; (*Контроль напряжения силового шкафа*)
	DM_D3 AT %IX9.11.0.0.2:BOOL (*Давление масла*);
	TM_D3 AT %IW9.2.0.0: WORD; (*Контроль температуры масла*)
	TZD3_D3 AT %IX9.11.0.0.5: BOOL; (*Тепловая защита контактора дробилки*)
	avto_D3 AT %IX9.11.0.0.6: BOOL; (*Выбор режима "автомат"*)
	RD3_D3 AT %IX9.11.0.0.7: BOOL; (*Контроль работы дробилки*)
	D3_mod2_byte AT %QW9.11.1.0 :BYTE; (*Битовая маска управления вторым модулем вх/вых дробилки Д3*)

	ready_D3 AT %QX3.1.2: BOOL; (*Готовность шкафа*)
	work_D3: BOOL; (*Команда разрешающая запуск следующей ступени*)
	nasos_D3: BOOL; (*Включение контактора насоса*)
	vent_D3: BOOL; (*Включение контактора вентилятора*)
	ten_D3: BOOL; (*Включение контактора ТЭНа*)
	KM1_D3: BOOL; (*Пуск основного контактора*)
	KM2_D3: BOOL; (*Запуск двигателя в "звезду"*)
	KM3_D3: BOOL; (*Основной пуск двигателя в "треугольник"*)
	out_avto_D3:BOOL; (*Переключение перекидного реле в режим автомат*)
	TM_D3_bool: BOOL;

	(*Дробилка Д4*)
	D4: D4;
	KU_D4 AT %IX9.12.0.0.0: BOOL; (*Контроль напряжения*)
	TZN_D4 AT %IX9.12.0.0.1: BOOL; (*Тепловая защита насоса*)
	UM_D4 AT %IX9.12.0.0.2: BOOL;  (*Уровень масла в маслостанции*)
	KPM_D4 AT %IX9.12.0.0.4: BOOL; (*Контроль протока масла*)
	TZV_D4 AT %IX9.12.0.0.5: BOOL; (*Тепловая защита вентилятора*)
	RMS_D4 AT %IX9.12.0.0.7: BOOL; (*Контроль работы насоса*)
	D4_mod1_byte AT %QW9.12.1.0 :BYTE (*Битовая маска управления первым модулем вх/вых дробилки Д4*);

	KUD3_D4 AT %IX9.13.0.0.0: BOOL; (*Контроль напряжения*)
	DM_D4 AT %IX9.13.0.0.2:BOOL (*Давление масла*);
	TM_D4 AT %IW9.1.0.0: WORD; (*Контроль температуры масла*)
	TZD3_D4 AT %IX9.13.0.0.5: BOOL; (*Тепловая защита контактора дробилки*)
	avto_D4 AT %IX9.13.0.0.6: BOOL; (*Выбор режима "автомат"*)
	RD3_D4 AT %IX9.13.0.0.7: BOOL; (*Контроль работы дробилки*)
	D4_mod2_byte AT %QW9.13.1.0 :BYTE (*Битовая маска управления вторым модулем вх/вых дробилки Д4*);

	ready_D4 AT %QX3.1.4: BOOL; (*Готовность шкафа*)
	work_D4: BOOL; (*Команда разрешающая запуск следующей ступени*)
	nasos_D4: BOOL; (*Включение контактора насоса*)
	vent_D4: BOOL; (*Включение контактора вентилятора*)
	ten_D4: BOOL; (*Включение контактора ТЭНа*)
	KM1_D4: BOOL; (*Пуск основного контактора*)
	KM2_D4: BOOL; (*Запуск двигателя в "звезду"*)
	KM3_D4: BOOL; (*Основной пуск двигателя в "треугольник"*)
	out_avto_D4:BOOL; (*Переключение перекидного реле в режим автомат*)
	TM_D4_bool: BOOL;

	work_level_10: BOOL;

(*Ленточный конвеер ЛК-10*)
	LK10: LK1;
	KU_LK10 AT %IX7.1.0.0.0: BOOL; (*Контроль напряжения*)
	TZ_LK10 AT %IX7.1.0.0.1: BOOL; (*Тепловая защита контактора*)
	tros_LK10 AT %IX7.1.0.0.2: BOOL; (*Тросовое ограждение*)
	VL_LK10 AT %IW7.1.2.0: WORD; (*Контроль скорости*)
	shod_LK10 AT %IX7.1.0.0.4: BOOL; (*Сход конвеерной ленты*)
	ogr_LK10 AT %IX7.1.0.0.5: BOOL; (*Защитное ограждение*)
	avto_LK10 AT %IX7.1.0.0.6: BOOL; (*Выбор режима "автомат"*)
	P_LK10 AT %IX7.1.0.0.7: BOOL; (*Контроль работы пускателя*)
	KM1_LK10  AT %QW7.1.1.0: BOOL; (*Включение пускателя*)

	ready_LK10 AT %QX2.3: BOOL; (*Готовность шкафа*)
	work_LK10: BOOL; (*Команда разрешающая запуск следующей ступени*)
 	ton_lk10:TON; (*задержка пуска конвеера*)
	counter_LK10: counter;  (*Счетчик импульсов, для оределения скорости вращения*)
	bool_Vl_LK10: BOOL; (*Подтверждение скорости вращения*)

(*Ленточный конвеер ЛК-11*)
	LK11: LK1;
	KU_LK11 AT %IX7.2.0.0.0: BOOL; (*Контроль напряжения*)
	TZ_LK11 AT %IX7.2.0.0.1: BOOL; (*Тепловая защита контактора*)
	tros_LK11 AT %IX7.2.0.0.2:BOOL; (*Тросовое ограждение*)
	VL_LK11 AT %IW7.2.2.0: WORD; (*Контроль скорости*)
	shod_LK11 AT %IX7.2.0.0.4: BOOL; (*Сход конвеерной ленты*)
	ogr_LK11 AT %IX7.2.0.0.5: BOOL; (*Защитное ограждение*)
	avto_LK11 AT %IX7.2.0.0.6: BOOL; (*Выбор режима "автомат"*)
	P_LK11 AT %IX7.2.0.0.7: BOOL; (*Контроль работы пускателя*)
	KM1_LK11 AT %QW7.2.1.0: BOOL; (*Включение пускателя*)

	ready_LK11 AT %QX3.0.0: BOOL; (*Готовность шкафа*)
	work_LK11: BOOL; (*Команда разрешающая запуск следующей ступени*)
	ton_lk11:TON; (*задержка пуска конвеера*)
	counter_LK11: counter;  (*Счетчик импульсов, для оределения скорости вращения*)
	bool_Vl_LK11: BOOL; (*Подтверждение скорости вращения*)

(*Ленточный конвеер ЛК-12*)
	LK12: LK12_modern;
	KU_LK12 AT %IX7.3.0.0.0: BOOL; (*Контроль напряжения*)
	TZ_LK12 AT %IX7.3.0.0.1: BOOL; (*Тепловая защита контактора*)
	tros_LK12 AT %IX7.3.0.0.2: BOOL; (*Тросовое ограждение*)
	VL_LK12 AT %IW7.3.2.0: WORD; (*Контроль скорости*)
	shod_LK12 AT %IX7.3.0.0.4: BOOL; (*Сход конвеерной ленты*)
	ogr_LK12 AT %IX7.3.0.0.5: BOOL; (*Защитное ограждение*)
	avto_LK12 AT %IX7.3.0.0.6: BOOL; (*Выбор режима "автомат"*)
	P_LK12 AT %IX7.3.0.0.7: BOOL; (*Контроль работы пускателя*)
	KM1_LK12 AT %QW7.3.1.0: BOOL; (*Включение пускателя*)

	ready_LK12  AT %QX3.0.1: BOOL; (*Готовность шкафа*)
	work_LK12: BOOL; (*Команда разрешающая запуск следующей ступени*)
	ton_lk12:TON; (*задержка пуска конвеера*)
	counter_LK12: counter;  (*Счетчик импульсов, для оределения скорости вращения*)
	bool_Vl_LK12: BOOL; (*Подтверждение скорости вращения*)

(*Ленточный конвеер ЛК-13*)
	LK13: LK1;
	KU_LK13 AT %IX7.4.0.0.0: BOOL; (*Контроль напряжения*)
	TZ_LK13 AT %IX7.4.0.0.1: BOOL; (*Тепловая защита контактора*)
	tros_LK13 AT %IX7.4.0.0.2: BOOL; (*Тросовое ограждение*)
	VL_LK13 AT %IW7.4.2.0: WORD; (*Контроль скорости*)
	shod_LK13 AT %IX7.4.0.0.4: BOOL; (*Сход конвеерной ленты*)
	ogr_LK13 AT %IX7.4.0.0.5: BOOL; (*Защитное ограждение*)
	avto_LK13 AT %IX7.4.0.0.6: BOOL; (*Выбор режима "автомат"*)
	P_LK13 AT %IX7.4.0.0.7: BOOL; (*Контроль работы пускателя*)
	KM1_LK13 AT %QW7.4.1.0: BOOL; (*Включение пускателя*)

	ready_LK13  AT %QX3.0.2: BOOL; (*Готовность шкафа*)
	work_LK13: BOOL; (*Команда разрешающая запуск следующей ступени*)
	ton_lk13:TON; (*задержка пуска конвеера*)
	counter_LK13: counter;  (*Счетчик импульсов, для оределения скорости вращения*)
	bool_Vl_LK13: BOOL; (*Подтверждение скорости вращения*)

	work_level_1: BOOL;

	(*Грохот ГР-3*)
	GR3: Grohot;
	KU_GR3 AT %IX7.5.0.0.0: BOOL; (*Контроль напряжения*)
	TZ_GR3 AT %IX7.5.0.0.1: BOOL; (*Тепловая защита контактора*)
	STOP_GR3 AT %IX7.5.0.0.2: BOOL (*грибок ГР3*);
	avto_GR3 AT %IX7.5.0.0.6: BOOL; (*Выбор режима "автомат"*)
	P_GR3 AT %IX7.5.0.0.7: BOOL; (*Контроль работы пускателя*)
	KM1_GR3 AT %QW7.5.1.0: BOOL; (*Включение пускателя*)

	ready_GR3 AT %QX3.0.3: BOOL; (*Готовность шкафа*)
	work_GR3: BOOL; (*Команда разрешающая запуск следующей ступени*)
	ton_GR3:TON; (*задержка пуска грохота*)

	work_level_2: BOOL;

	(*Ленточный конвеер ЛК-7*)
	LK7: LK3;
	KU_LK7 AT %IX9.5.0.0.0: BOOL; (*Контроль напряжения*)
	TZ_LK7 AT %IX9.5.0.0.1: BOOL; (*Тепловая защита контактора*)
	tros_LK7 AT %IX9.5.0.0.2: BOOL; (*Тросовое ограждение*)
	VL_LK7 AT %IW9.5.2.0: WORD; (*Контроль скорости*)
	shod_LK7 AT %IX9.5.0.0.4: BOOL; (*Сход конвеерной ленты*)
	ogr_LK7 AT %IX9.5.0.0.5: BOOL; (*Защитное ограждение*)
	avto_LK7 AT %IX9.5.0.0.6: BOOL; (*Выбор режима "автомат"*)
	P_LK7 AT %IX9.5.0.0.7:BOOL; (*Контроль работы пускателя*)
	KM1_LK7 AT %QW9.5.1.0: BOOL; (*Включение пускателя*)

	ready_LK7 AT %QX3.0.4: BOOL; (*Готовность шкафа*)
	work_LK7: BOOL; (*Команда разрешающая запуск следующей ступени*)
	ton_LK7:TON; (*задержка пуска конвеера*)
	counter_LK7: counter_lk5;  (*Счетчик импульсов, для оределения скорости вращения*)
	bool_Vl_LK7: BOOL; (*Подтверждение скорости вращения*)

	(*Ленточный конвеер ЛК-8*)
	LK8: LK1;
	KU_LK8 AT %IX9.6.0.0.0: BOOL; (*Контроль напряжения*)
	TZ_LK8 AT %IX9.6.0.0.1: BOOL; (*Тепловая защита контактора*)
	tros_LK8 AT %IX9.6.0.0.2: BOOL; (*Тросовое ограждение*)
	VL_LK8 AT %IW9.6.2.0: WORD; (*Контроль скорости*)
	shod_LK8 AT %IX9.6.0.0.4: BOOL; (*Сход конвеерной ленты*)
	ogr_LK8 AT %IX9.6.0.0.5: BOOL; (*Защитное ограждение*)
	avto_LK8 AT %IX9.6.0.0.6: BOOL; (*Выбор режима "автомат"*)
	P_LK8 AT %IX9.6.0.0.7:BOOL; (*Контроль работы пускателя*)
	KM1_LK8 AT %QW9.6.1.0: BOOL; (*Включение пускателя*)

	ready_LK8 AT %QX3.0.5: BOOL; (*Готовность шкафа*)
	work_LK8: BOOL; (*Команда разрешающая запуск следующей ступени*)
	ton_LK8:TON; (*задержка пуска конвеера*)
	ton_LK81:TON; (*задержка пуска конвеера*)
	counter_LK8: counter_lk5;  (*Счетчик импульсов, для оределения скорости вращения*)
	bool_Vl_LK8: BOOL; (*Подтверждение скорости вращения*)

	(*Ленточный конвеер ЛК-6*)
	LK6: LK3;
	KU_LK6 AT %IX7.6.0.0.0: BOOL; (*Контроль напряжения*)
	TZ_LK6 AT %IX7.6.0.0.1: BOOL; (*Тепловая защита контактора*)
	tros_LK6 AT %IX7.6.0.0.2: BOOL; (*Тросовое ограждение*)
	VL_LK6 AT %IW7.6.2.0: WORD; (*Контроль скорости*)
	shod_LK6 AT %IX7.6.0.0.4: BOOL; (*Сход конвеерной ленты*)
	ogr_LK6 AT %IX7.6.0.0.5: BOOL; (*Защитное ограждение*)
	avto_LK6 AT %IX7.6.0.0.6: BOOL; (*Выбор режима "автомат"*)
	P_LK6 AT %IX7.6.0.0.7:BOOL;  (*Контроль работы пускателя*)
	KM1_LK6 AT %QW7.6.1.0: BOOL; (*Включение пускателя*)

	ready_LK6 AT %QX3.0.7: BOOL; (*Готовность шкафа*)
	work_LK6: BOOL; (*Команда разрешающая запуск следующей ступени*)
	ton_LK6:TON; (*задержка пуска конвеера*)
	counter_LK6: counter;  (*Счетчик импульсов, для оределения скорости вращения*)
	bool_Vl_LK6: BOOL; (*Подтверждение скорости вращения*)

	(*Ленточный конвеер ЛК-9*)
	LK9: LK1;
	KU_LK9 AT %IX7.7.0.0.0: BOOL; (*Контроль напряжения*)
	TZ_LK9 AT %IX7.7.0.0.1: BOOL; (*Тепловая защита контактора*)
	tros_LK9 AT %IX7.7.0.0.2: BOOL; (*Тросовое ограждение*)
	VL_LK9 AT %IW7.7.2.0: WORD; (*Контроль скорости*)
	shod_LK9 AT %IX7.7.0.0.4: BOOL; (*Сход конвеерной ленты*)
	ogr_LK9 AT %IX7.7.0.0.5: BOOL; (*Защитное ограждение*)
	avto_LK9 AT %IX7.7.0.0.6: BOOL; (*Выбор режима "автомат"*)
	P_LK9 AT %IX7.7.0.0.7:BOOL;  (*Контроль работы пускателя*)
	KM1_LK9 AT %QW7.7.1.0: BOOL; (*Включение пускателя*)

	ready_LK9 AT %QX3.0.6: BOOL; (*Готовность шкафа*)
	work_LK9: BOOL; (*Команда разрешающая запуск следующей ступени*)
	ton_LK9:TON; (*задержка пуска конвеера*)
	counter_LK9: counter;  (*Счетчик импульсов, для оределения скорости вращения*)
	bool_Vl_LK9: BOOL; (*Подтверждение скорости вращения*)

	work_level_3: BOOL;

 (*Шкаф ленточного питателя №1-№3*)
	LP1_3: LP1_3;
	Vl1_LP1_3 AT %IW7.9.2.0: WORD; (*Контроль скорости ЛП1*)
	Vl2_LP1_3 AT %IW7.9.3.0: WORD; (*Контроль скорости ЛП2*)
	Vl3_LP1_3 AT %IW7.9.4.0: WORD; (*Контроль скорости ЛП3*)
	stop2_LP1_3 AT %IX7.9.0.0.3: BOOL; (*грибок ЛП1_3*)
	KM2345_LP1_3_byte AT %QW7.9.1.0: BYTE; (*Пуск контакторов через РС, с помощью пакования в байт*)


	in_020 AT %IX1.0.1: BOOL; (*Выбор размера фракции: 0-20мм*)
	in_040 AT %IX1.0.2: BOOL; (*Выбор размера фракции: 0-40мм*)
	in_020_4070 AT %IX1.0.3: BOOL; (*Выбор размера фракции: 0-20мм и 40-70мм*)
	ready_LP1_3 AT %QX3.1.0: BOOL; (*Готовность шкафа*)

	KU_LP1_3 AT %IX7.8.0.0.0: BOOL; (*Контроль напряжения*)
	TZ1_LP1_3 AT %IX7.8.0.0.1: BOOL; (*Тепловая защита контактора ЛП1*)
	TZ2_LP1_3 AT %IX7.8.0.0.2: BOOL; (*Тепловая защита контактора ЛП2*)
	TZ3_LP1_3 AT %IX7.8.0.0.3: BOOL; (*Тепловая защита контактора ЛП3*)
	PRO_LP1_3 AT %IX7.8.0.0.4: BOOL; (*Положение рабочего органа*)
	avto_LP1_3 AT %IX7.8.0.0.6: BOOL; (*Выбор режима "автомат"*)
	P_LP1_3 AT %IX7.8.0.0.7:BOOL;  (*Контроль работы пускателя*)
	KM1_LP1_3 AT %QW7.8.1.0 :BOOL; (*Включение пускателя ЛП1*)

	KM2_LP1_3 :BOOL; (*Включение пускателя ЛП2 - вправо*)
	KM4_LP1_3 :BOOL; (*Включение пускателя ЛП3 - вправо*)
	KM5_LP1_3 :BOOL; (*Включение пускателя ЛП3 - влево*)
	KM3_LP1_3 :BOOL; (*Включение пускателя ЛП2 - влево*)
	work_LP1_3: BOOL; (*Команда разрешающая запуск следующей ступени*)
	ton_LP1_3:TON; (*Задержка времени пуска ленточного питателя 1-3*)
	counter_LP1_3_1: counter;   (*Счетчик импульсов, для оределения скорости вращения*)
	bool_Vl1_LP1_3: BOOL; (*Подтверждение скорости вращения*)
	counter_LP1_3_2: counter;  (*Счетчик импульсов, для оределения скорости вращения*)
	bool_Vl2_LP1_3: BOOL; (*Подтверждение скорости вращения*)
	counter_LP1_3_3: counter;  (*Счетчик импульсов, для оределения скорости вращения*)
	bool_Vl3_LP1_3: BOOL; (*Подтверждение скорости вращения*)

	(*Грохот ГР-2*)
	GR2: Grohot1;
	KU_GR2 AT %IX7.10.0.0.0: BOOL; (*Контроль напряжения*)
	TZ_GR2 AT %IX7.10.0.0.1: BOOL; (*Тепловая защита контактора*)
	STOP_GR2 AT %IX7.10.0.0.2: BOOL;(*грибок ГР2*)
	avto_GR2 AT %IX7.10.0.0.6: BOOL; (*Выбор режима "автомат"*)
	P_GR2 AT %IX7.10.0.0.7:BOOL;  (*Контроль работы пускателя*)
	KM1_GR2 AT %QW7.10.1.0: BOOL; (*Включение пускателя*)

	ready_GR2  AT %QX3.1.1: BOOL; (*Готовность шкафа*)
	work_GR2: BOOL; (*Команда разрешающая запуск следующей ступени*)
	ton_GR2:TON; (*Задержка времени пуска грохота 2*)

	work_level_4: BOOL;

	(*Ленточный конвеер ЛК-5*)
	LK5: LK1;
	KU_LK5 AT %IX9.7.0.0.0: BOOL; (*Контроль напряжения*)
	TZ_LK5 AT %IX9.7.0.0.1: BOOL; (*Тепловая защита контактора*)
	tros_LK5 AT %IX9.7.0.0.2: BOOL; (*Тросовое ограждение*)
	VL_LK5 AT %IW9.7.2.0: WORD; (*Контроль скорости*)
	shod_LK5 AT %IX9.7.0.0.4: BOOL; (*Сход конвеерной ленты*)
	ogr_LK5 AT %IX9.7.0.0.5: BOOL; (*Защитное ограждение*)
	avto_LK5 AT %IX9.7.0.0.6: BOOL; (*Выбор режима "автомат"*)
	P_LK5 AT %IX9.7.0.0.7: BOOL; (*Контроль работы пускателя*)
	KM1_LK5 AT %QW9.7.1.0: BOOL; (*Включение контактора*)

	ready_LK5 AT %QX3.1.3: BOOL; (*Готовность шкафа*)
	work_LK5: BOOL; (*Команда разрешающая запуск следующей ступени*)
	ton_lk5:TON; (*задержка пуска конвеера*)
	counter_lk5: counter_lk5;  (*Счетчик импульсов, для оределения скорости вращения*)
	bool_Vl_LK5: BOOL; (*Подтверждение скорости вращения*)

	work_level_6: BOOL;
	work_level_61: BOOL;

(*Ленточный питатель ЛП-4*)
	LP4: LP4_without_FC;
	KU_LP4 AT %IX9.8.0.0.0: BOOL; (*контроль напряжения*)
	TZ_LP4 AT %IX9.8.0.0.1: BOOL; (*срабатывание тепловой защиты двигателя*)
	MD2_LP4 AT %IX9.8.0.0.5: BOOL; (*срабаьывание металлдетектора*)
	avto_LP4 AT %IX9.8.0.0.6: BOOL; (*Выбор режима "автомат"*)
	P_LP4 AT %IX9.8.0.0.7: BOOL; (*контроль реботы шкафа*)
	KM1_LP4 AT %QW9.8.1.0: BOOL; (*включение контактора*)

	ready_LP4  AT %QX3.1.6: BOOL; (*готовность шкафа*)
	work_LP4: BOOL; (*команда разрешающая пуск следующей ступени*)
	metall_LP4: BOOL; (*срабаьывание металлдетектора*)

(*Ленточный питатель ЛП5*)
	LP5: LP5;
	avto_out_LP5 AT %QW9.9.1.0: BOOL; (*Переключение реле в режим "автомат"*)
	STOP_LP5 AT %IX9.9.0.0.2: BOOL (*грибок ЛП5*);
	VL_LP5: WORD; (*контроль скорости ленты*)
	MD2_LP5 AT %IX9.9.0.0.5: BOOL; (*срабаьывание металлдетектора*)
	avto_LP5 AT %IX9.9.0.0.6: BOOL; (*Выбор режима "автомат"*)
	avar_FC_LP5 AT %IX9.9.0.0.0: BOOL;

	ready_LP5 AT %QX3.1.7: BOOL; (*готовность шкафа*)
	work_LP5: BOOL; (*команда разрешающая пуск следующей ступени*)
	metall_LP5: BOOL; (*срабаьывание металлдетектора*)
	counter_LP5: counter;  (*Счетчик импульсов, для оределения скорости вращения*)
	bool_Vl_LP5: BOOL; (*Подтверждение скорости вращения*)

	pusk_LP5 AT %QW9.4.0.0: WORD; (*каманда на пуск частотника*)
	b1_00_LP5 AT %QW9.4.1.0: WORD; (*Команда на изменение режима частотника: управление частотой с помощью компьютера*)
	b1_04_LP5 AT %QW9.4.2.0: WORD;	(*Команда на изменение режима частотника: разрешение на установку частоты с компьютера*)
	output_Hz_LP5 AT %IW9.4.3.0: WORD; (*Выходная частота*)
	in_P_LP5 AT %IW9.4.4.0: WORD; (*Индикатор работы частотника ЛП5*)

(*Ленточный конвеер ЛК-4*)
	LK4: LK4;
	ton_LK4: TON; (*задержка времени пуска*)
	KU_LK4 AT %IX7.11.0.0.0: BOOL; (*контроль напряжения*)
	TZ_LK4 AT %IX7.11.0.0.1: BOOL; (*срабатывание тепловой защиты двигателя*)
	tros_LK4 AT %IX7.11.0.0.2: BOOL; (*тросовое ограждение*)
	VL_LK4 AT %IW7.11.2.0: WORD; (*контроль скорости ленты*)
	shod_LK4 AT %IX7.11.0.0.4: BOOL; (*сход лениы*)
	MD3_LK4 AT %IX7.11.0.0.5: BOOL; (*срабатывание металлдетектора*)
	avto_LK4 AT %IX7.11.0.0.6: BOOL; (*выбор режима "автомат"*)
	P_LK4 AT %IX7.11.0.0.7: BOOL; (*контроль реботы шкафа*)
	KM1_LK4 AT %QW7.11.1.0: BOOL; (*включение контактора*)

	ready_LK4 AT %QX3.2.1: BOOL; (*готовность шкафа*)
	work_LK4: BOOL; (*команда разрешающая пуск следующей ступени*)
	counter_LK4: counter;  (*Счетчик импульсов, для оределения скорости вращения*)
	bool_Vl_LK4: BOOL; (*Подтверждение скорости вращения*)
	metall_LK4: BOOL; (*срабатывание металлдетектора*)

(*Грохот ГР-1*)
	GR1: Grohot;
	ton_GR1: TON; (*задержка времени пуска*)

	KU_GR1 AT %IX7.12.0.0.0: BOOL; (*контроль напряжения*)
	TZ_GR1 AT %IX7.12.0.0.1: BOOL; (*срабатывание тепловой защиты двигателя*)
	STOP_GR1 AT %IX7.12.0.0.2: BOOL (*грибок ГР1*);
	avto_GR1 AT %IX7.12.0.0.6: BOOL; (*выбор режима "автомат"*)
	P_GR1 AT %IX7.12.0.0.7: BOOL; (*контроль срабатывания пускателя*)
	KM1_GR1 AT %QW7.12.1.0: BOOL; (*включение контактора*)

	ready_GR1 AT %QX3.2.0: BOOL; (*готовность шкафа*)
	work_GR1: BOOL; (*разрешение на работу следующей ступени*)

(*Ленточный конвеер ЛК-2*)
	LK2: LK2;
	KU_LK2 AT %IX7.13.0.0.0: BOOL; (*контроль напряжения*)
	TZ_LK2 AT %IX7.13.0.0.1: BOOL; (*срабатывание тепловой защиты двигателя*)
	tros_LK2 AT %IX7.13.0.0.2: BOOL; (*тросовая защита*)
	shod_LK2 AT %IX7.13.0.0.4: BOOL; (*сход ленты*)
	ogr_LK2 AT %IX7.13.0.0.5: BOOL; (*ограждение*)
	avto_LK2 AT %IX7.13.0.0.6: BOOL; (*выбор режима "автомат"*)
	P_LK2 AT %IX7.13.0.0.7: BOOL; (*контроль работы пускателя*)
	LK2_out AT %QW7.13.1.0: BYTE (*управление битовой маской выходов*);
	ready_LK2 AT %QX3.2.2: BOOL; (*готовность шкафа*)
	Vl_LK2 AT %IW7.13.2.0: WORD;

	KM1_LK2: BOOL; (*пуск контактора*)
	work_LK2: BOOL; (*разрешение на работу следующей ступени*)
	ton_LK2: TON; (*задержка времени пуска*)
	counter_LK2: counter;  (*Счетчик импульсов, для оределения скорости вращения*)
	bool_Vl_LK2: BOOL; (*Подтверждение скорости вращения*)

(*Ленточный конвеер ЛК-3*)
	LK3: LK1;
	KU_LK3 AT %IX7.14.0.0.0: BOOL; (*контроль напряжения*)
	TZ_LK3 AT %IX7.14.0.0.1: BOOL; (*срабатывание тепловой защиты*)
	tros_LK3 AT %IX7.14.0.0.2: BOOL; (*троссовая защита*)
	VL_LK3 AT %IW7.14.2.0: WORD; (*контроль скорости лентыя*)
	shod_LK3 AT %IX7.14.0.0.4: BOOL; (*сход лениты*)
	ogr_LK3 AT %IX7.14.0.0.5: BOOL; (*ограждение*)
	avto_LK3 AT %IX7.14.0.0.6: BOOL; (*выбор режима "автомат"*)
	P_LK3 AT %IX7.14.0.0.7: BOOL; (*контроль работы пускаьтеля*)
	KM1_LK3 AT %QW7.14.1.0: BOOL; (*пуск контактора*)

	ready_LK3 AT %QX2.0: BOOL; (*готовность шкафа*)
	work_LK3: BOOL; (*разрешение на работу следующей ступени*)
	ton_LK3: TON; (*задержка времени пуска*)
	counter_LK3: counter;  (*Счетчик импульсов, для оределения скорости вращения*)
	bool_Vl_LK3: BOOL; (*Подтверждение скорости вращения*)

(*Вибропитатель ВП-1*)
	VP1: VP1;
	KU_VP1 AT %IX7.15.0.0.0:BOOL; (*контроль напряжения после автомата*)
	TZ_VP1 AT %IX7.15.0.0.1:BOOL; (*срабатывание тепловой защиты*)
	stop_VP1 AT %IX7.15.0.0.2: BOOL (*грибок ВП1*);
	avto_VP1 AT %IX7.15.0.0.6: BOOL; (*выбор режима "автомат"*)
	P_VP1 AT %IX7.15.0.0.7: BOOL;
	pusk_VP1 AT %QW7.15.1.0: BOOL; (*Команда на ВП1*)

	ready_VP1 AT %QX3.2.3: BOOL; (*готовность шкафа*)
	work_VP1: BOOL; (*разрешение на пуск следующей ступени*)

	stop_VP1_LK7: stop_VP1;
	LV_LK7 AT %ID9.3.0.0: REAL; (*Входной сигнал от датчика наполнения бункера ЛК7*)
	LV_low_LK7: BOOL; (*первый уровень бункера ЛК7*)
	LV_high_LK7: BOOL; (*второй уровень бункера ЛК7*)

	stop_VP1_LK8: stop_VP1;
	LV_LK8 AT %ID9.3.1.0:REAL; (*Входной сигнал от датчика наполнения бункера ЛК8*)
	LV_low_LK8: BOOL; (*первый уровень бункера ЛК8*)
	LV_high_LK8: BOOL; (*второй уровень бункера ЛК8*)

	stop_VP1_D2: stop_VP1;
	LV_D2 AT %ID7.18.0.0: REAL; (*Входной сигнал от датчика наполнения дробилки Д2*)
	LV_low_D2: BOOL; (*первый уровень дробилки Д2*)
	LV_high_D2: BOOL; (*первый уровень дробилки Д2*)

	LV_GR1 AT %ID7.18.1.0:REAL; (*входное значение уровня в бункере ГР1*)
	stop_PP1: stop_VP1;
	LV_low_GR1: BOOL; (*первый уровень бункера ГР1*)
	LV_high_GR1: BOOL; (*второй уровень бункера ГР1*)

	work_level_9: BOOL;

(*Блок вывода сигналов для SCADA*)
	signals: signals;
	KU_D2_out AT %QX8.1.0.0: BOOL;
	RMS_2_2_out AT %QX8.1.0.1: BOOL;
	avto_D2_out AT %QX8.1.0.2: BOOL;
	work_D2_out AT %QX8.1.0.3: BOOL;
	ready_D2_out AT %QX8.1.0.4: BOOL;
	TZD2_out AT %QX8.1.0.5: BOOL;
	KU_D3_out AT %QX8.1.0.6: BOOL;
	TZN_D3_out AT %QX8.1.0.7: BOOL;

	UM_D3_out AT %QX8.2.0.0: BOOL;
	KPM_D3_out AT %QX8.2.0.1: BOOL;
	TZV_D3_out AT %QX8.2.0.2: BOOL;
	avto_D3_out AT %QX8.2.0.3: BOOL;
	KUD3_D3_out AT %QX8.2.0.4: BOOL;
	TZD3_D3_out AT %QX8.2.0.5: BOOL;
	work_D3_out AT %QX8.2.0.6: BOOL;
	ready_D3_out AT %QX8.2.0.7: BOOL;

	TM_D3_out AT %QX8.3.0.0: BOOL;
	RMS_D3_out AT %QX8.3.0.1: BOOL;
	KU_D4_out AT %QX8.3.0.2: BOOL;
	TZN_D4_out AT %QX8.3.0.3: BOOL;
	UM_D4_out AT %QX8.3.0.4: BOOL;
	KPM_D4_out AT %QX8.3.0.5: BOOL;
	TZV_D4_out AT %QX8.3.0.6: BOOL;
	KUD3_D4_out AT %QX8.3.0.7: BOOL;

	TZD3_D4_out AT %QX8.4.0.0: BOOL;
	work_D4_out AT %QX8.4.0.1: BOOL;
	ready_D4_out AT %QX8.4.0.2: BOOL;
	avto_D4_out AT %QX8.4.0.3: BOOL;
	TM_D4_out AT %QX8.4.0.4: BOOL;
	RMS_D4_out AT %QX8.4.0.5: BOOL;
	KU_LK10_out AT %QX8.4.0.6: BOOL;
	TZ_LK10_out AT %QX8.4.0.7: BOOL;

	tros_LK10_out AT %QX8.5.0.0: BOOL;
	shod_LK10_out AT %QX8.5.0.1: BOOL;
	ogr_LK10_out AT %QX8.5.0.2: BOOL;
	TZ_LK12_out AT %QX8.5.0.3: BOOL;
	MD2_LP5_out AT %QX8.5.0.4: BOOL;
	avto_LK10_out AT %QX8.5.0.6: BOOL;
	ready_LK10_out AT %QX8.5.0.7: BOOL;

	work_LK10_out AT %QX8.6.0.0: BOOL;
	KU_LK11_out AT %QX8.6.0.1: BOOL;
	TZ_LK11_out AT %QX8.6.0.2: BOOL;
	tros_LK11_out AT %QX8.6.0.3: BOOL;
	shod_LK11_out AT %QX8.6.0.4: BOOL;
	ogr_LK11_out AT %QX8.6.0.5: BOOL;
	ato_LK11_out AT %QX8.6.0.6: BOOL;
	ready_LK11_out AT %QX8.6.0.7: BOOL;

	work_LK11_out AT %QX8.7.0.0: BOOL;
	KU_LK12_out AT %QX8.7.0.1: BOOL;
	tros_LK12_out AT %QX8.7.0.2: BOOL;
	shod_LK12_out AT %QX8.7.0.3: BOOL;
	ogr_LK12_out AT %QX8.7.0.4: BOOL;
	avto_LK12_out AT %QX8.7.0.5: BOOL;
	ready_LK12_out AT %QX8.7.0.6: BOOL;
	work_LK12_out AT %QX8.7.0.7: BOOL;

	KU_LK13_out AT %QX8.8.0.0: BOOL;
	TZ_LK13_out AT %QX8.8.0.1: BOOL;
	tros_LK13_out AT %QX8.8.0.2: BOOL;
	shod_LK13_out AT %QX8.8.0.3: BOOL;
	ogr_LK13_out AT %QX8.8.0.4: BOOL;
	avto_LK13_out AT %QX8.8.0.5: BOOL;
	ready_LK13_out AT %QX8.8.0.6: BOOL;
	work_LK13_out AT %QX8.8.0.7: BOOL;

	avto_GR3_out AT %QX8.9.0.0: BOOL;
	KU_GR3_out AT %QX8.9.0.1: BOOL;
	TZ_GR3_out AT %QX8.9.0.2: BOOL;
	ready_GR3_out AT %QX8.9.0.3: BOOL;
	work_GR3_out AT %QX8.9.0.4: BOOL;
	KU_LK7_out AT %QX8.9.0.5: BOOL;
	TZ_LK7_out AT %QX8.9.0.6: BOOL;
	tros_LK7_out AT %QX8.9.0.7: BOOL;

	shod_LK7_out AT %QX8.10.0.0: BOOL;
	ogr_LK7_out AT %QX8.10.0.1: BOOL;
	avto_LK7_out AT %QX8.10.0.2: BOOL;
	ready_LK7_out AT %QX8.10.0.3: BOOL;
	work_LK7_out AT %QX8.10.0.4: BOOL;
	KU_LK8_out AT %QX8.10.0.5: BOOL;
	TZ_LK8_out AT %QX8.10.0.6: BOOL;
	tros_LK8_out AT %QX8.10.0.7: BOOL;

	shod_LK8_out AT %QX8.11.0.0: BOOL;
	ogr_LK8_out AT %QX8.11.0.1: BOOL;
	avto_LK8_out AT %QX8.11.0.2: BOOL;
	ready_LK8_out AT %QX8.11.0.3: BOOL;
	work_LK8_out AT %QX8.11.0.4: BOOL;
	KU_LK6_out AT %QX8.11.0.5: BOOL;
	TZ_LK6_out AT %QX8.11.0.6: BOOL;
	tros_LK6_out AT %QX8.11.0.7: BOOL;

	shod_LK6_out AT %QX8.12.0.0: BOOL;
	ogr_LK6_out AT %QX8.12.0.1: BOOL;
	avto_LK6_out AT %QX8.12.0.2: BOOL;
	ready_LK6_out AT %QX8.12.0.3: BOOL;
	work_LK6_out AT %QX8.12.0.4: BOOL;
	KU_LK9_out AT %QX8.12.0.5: BOOL;
	TZ_LK9_out AT %QX8.12.0.6: BOOL;
	tros_LK9_out AT %QX8.12.0.7: BOOL;

	shod_LK9_out AT %QX8.13.0.0: BOOL;
	ogr_LK9_out AT %QX8.13.0.1: BOOL;
	avto_LK9_out AT %QX8.13.0.2: BOOL;
	ready_LK9_out AT %QX8.13.0.3: BOOL;
	work_LK9_out AT %QX8.13.0.4: BOOL;
	KU_LP1_3_out AT %QX8.13.0.5: BOOL;
	in_020_out AT %QX8.13.0.6: BOOL;
	in_040_out AT %QX8.13.0.7: BOOL;

	in_020_4070_out AT %QX8.14.0.0: BOOL;
	TZ1_LP1_3_out AT %QX8.14.0.1: BOOL;
	TZ2_LP1_3_out AT %QX8.14.0.2: BOOL;
	TZ3_LP1_3_out AT %QX8.14.0.3: BOOL;
	PRO_LP1_3_out AT %QX8.14.0.4: BOOL;
	avto_LP1_3_out AT %QX8.14.0.5: BOOL;
	ready_LP1_3_out AT %QX8.14.0.6: BOOL;
	work_LP1_3_out AT %QX8.14.0.7: BOOL;

	avto_GR2_out AT %QX8.15.0.0: BOOL;
	KU_GR2_out AT %QX8.15.0.1: BOOL;
	TZ_GR2_out AT %QX8.15.0.2: BOOL;
	ready_GR2_out AT %QX8.15.0.3: BOOL;
	work_GR2_out AT %QX8.15.0.4: BOOL;
	KU_LK5_out AT %QX8.15.0.5: BOOL;
	TZ_LK5_out AT %QX8.15.0.6: BOOL;
	tros_LK5_out AT %QX8.15.0.7: BOOL;

	shod_LK5_out AT %QX8.16.0.0: BOOL;
	ogr_LK5_out AT %QX8.16.0.1: BOOL;
	avto_LK5_out AT %QX8.16.0.2: BOOL;
	ready_LK5_out AT %QX8.16.0.3: BOOL;
	work_LK5_out AT %QX8.16.0.4: BOOL;
	KU_LK4_out AT %QX8.16.0.5: BOOL;
	TZ_LK4_out AT %QX8.16.0.6: BOOL;
	tros_LK4_out AT %QX8.16.0.7: BOOL;

	shod_LK4_out AT %QX8.17.0.0: BOOL;
	stop2_LP1_3_out AT %QX8.17.0.1: BOOL;
	avto_LK4_out AT %QX8.17.0.2: BOOL;
	ready_LK4_out AT %QX8.17.0.3: BOOL;
	work_LK4_out AT %QX8.17.0.4: BOOL;
	avto_GR1_out AT %QX8.17.0.5: BOOL;
	KU_GR1_out AT %QX8.17.0.6: BOOL;
	TZ_GR1_out AT %QX8.17.0.7: BOOL;

	ready_GR1_out AT %QX8.18.0.0: BOOL;
	work_GR1_out AT %QX8.18.0.1: BOOL;
	KU_LK2_out AT %QX8.18.0.2: BOOL;
	TZ_LK2_out AT %QX8.18.0.3: BOOL;
	tros_LK2_out AT %QX8.18.0.4: BOOL;
	shod_LK2_out AT %QX8.18.0.5: BOOL;
	ogr_LK2_out AT %QX8.18.0.6: BOOL;
	avto_LK2_out AT %QX8.18.0.7: BOOL;

	ready_LK2_out AT %QX8.19.0.0: BOOL;
	work_LK2_out AT %QX8.19.0.1: BOOL;
	KU_LK3_out AT %QX8.19.0.2: BOOL;
	TZ_LK3_out AT %QX8.19.0.3: BOOL;
	tros_LK3_out AT %QX8.19.0.4: BOOL;
	shod_LK3_out AT %QX8.19.0.5: BOOL;
	ogr_LK3_out AT %QX8.19.0.6: BOOL;
	avto_LK3_out AT %QX8.19.0.7: BOOL;

	ready_LK3_out AT %QX8.20.0.0: BOOL;
	work_LK3_out AT %QX8.20.0.1: BOOL;
	avto_LP4_out AT %QX8.20.0.2: BOOL;
	ready_LP4_out AT %QX8.20.0.3: BOOL;
	work_LP4_out AT %QX8.20.0.4: BOOL;
	avto_LP5_out AT %QX8.20.0.5: BOOL;
	ready_LP5_out AT %QX8.20.0.6: BOOL;
	work_LP5_out AT %QX8.20.0.7: BOOL;

	avto_VP1_out AT %QX8.21.0.0: BOOL;
	ready_VP1_out AT %QX8.21.0.1: BOOL;
	work_VP1_out AT %QX8.21.0.2: BOOL;
	STOP_LP4_out AT %QX8.21.0.5: BOOL;
	STOP_LP5_out AT %QX8.21.0.6: BOOL;
	STOP_VP1_out AT %QX8.21.0.7: BOOL;

	DM_D3_out AT %QX8.22.0.0: BOOL;
	DM_D4_out AT %QX8.22.0.1: BOOL;
	STOP_GR3_out AT %QX8.22.0.2: BOOL;
	STOP_GR2_out AT %QX8.22.0.3: BOOL;
	STOP_GR1_out AT %QX8.22.0.4: BOOL;
	MD3_LK4_out AT %QX8.22.0.5: BOOL;
	PP1_out AT %QX8.22.0.6: BOOL;
	MD2_LP4_out AT %QX8.22.0.7: BOOL;

	avar_D2 AT %QX8.23.0.0: BOOL;
	avar_D3 AT %QX8.23.0.1: BOOL;
	avar_D4 AT %QX8.23.0.2: BOOL;
	avar_LK10 AT %QX8.23.0.3: BOOL;
	avar_LK11 AT %QX8.23.0.4: BOOL;
	avar_LK12 AT %QX8.23.0.5: BOOL;
	avar_LK13 AT %QX8.23.0.6: BOOL;
	avar_GR3 AT %QX8.23.0.7: BOOL;

	avar_LK7 AT %QX8.24.0.0: BOOL;
	avar_LK8 AT %QX8.24.0.1: BOOL;
	avar_LK6 AT %QX8.24.0.2: BOOL;
	avar_LK9 AT %QX8.24.0.3: BOOL;
	avar_LP1_3 AT %QX8.24.0.4: BOOL;
	avar_GR2 AT %QX8.24.0.5: BOOL;
	avar_LK5 AT %QX8.24.0.6: BOOL;
	avar_LP4 AT %QX8.24.0.7: BOOL;

	avar_LP5 AT %QX8.25.0.0: BOOL;
	avar_GR1 AT %QX8.25.0.1: BOOL;
	avar_LK4 AT %QX8.25.0.2: BOOL;
	avar_LK2 AT %QX8.25.0.3: BOOL;
	avar_VP1 AT %QX8.25.0.4: BOOL;
	avar_LK3 AT %QX8.25.0.5: BOOL;
	avto_all_out AT %QX8.25.0.6: BOOL;
	pusk_out AT %QX8.25.0.7: BOOL;

(*Блок аварийной остановки агрегатов, в случае отсутствия сигналов связи от них*)
	alarm: alarm;
	adr_dev_rs2 AT %QD7.0: DWORD;
	err_dev_rs2 AT %QW7.1: WORD;
	adr_dev_rs1 AT %QD9.0: DWORD;
	err_dev_rs1 AT %QW9.1: WORD;
	e_LK10_out AT %QX8.26.0.0: BOOL;
	e_LK11_out AT %QX8.26.0.1: BOOL;
	e_LK12_out AT %QX8.26.0.2: BOOL;
	e_LK13_out AT %QX8.26.0.3: BOOL;
	e_GR3_out AT %QX8.26.0.4: BOOL;
	e_LK7_out AT %QX8.26.0.5: BOOL;
	e_LK8_out AT %QX8.26.0.6: BOOL;
	e_LK6_out AT %QX8.26.0.7: BOOL;

	e_LK9_out AT %QX8.27.0.0: BOOL;
	e_LP13mod1_out AT %QX8.27.0.1: BOOL;
	e_LP13mod2_out AT %QX8.27.0.2: BOOL;
	e_GR2_out AT %QX8.27.0.3: BOOL;
	e_LK5_out AT %QX8.27.0.4: BOOL;
	e_LP4_out AT %QX8.27.0.5: BOOL;
	e_LP5_out AT %QX8.27.0.6: BOOL;
	e_LK4_out AT %QX8.27.0.7: BOOL;

	e_GR1_out AT %QX8.28.0.0: BOOL;
	e_LK2_out AT %QX8.28.0.1: BOOL;
	e_LK3_out AT %QX8.28.0.2: BOOL;
	e_VP1_out AT %QX8.28.0.3: BOOL;
	e_D3mod1_out AT %QX8.28.0.4: BOOL;
	e_D3mod2_out AT %QX8.28.0.5: BOOL;
	e_D4mod1_out AT %QX8.28.0.6: BOOL;
	e_D4mod2_out AT %QX8.28.0.7: BOOL;

	e_D2_out AT %QX8.29.0.0: BOOL;
	e_cyc1_out AT %QX8.29.0.1: BOOL;
	e_cyc2_out AT %QX8.29.0.2: BOOL;
	shnek_up_cyc_out AT %QX8.29.0.3: BOOL;
	avar_cyc_out AT %QX8.29.0.5: BOOL;


	lev_up_cyc_out AT %QX8.30.0.0: BOOL;
	pre_cyc_out AT %QX8.30.0.1: BOOL;
	ku_cyc_out AT %QX8.30.0.2: BOOL;
	tz_cyc_out AT %QX8.30.0.3: BOOL;
	ready_cyc_out AT %QX8.30.0.4: BOOL;
	work_cyc_out AT %QX8.30.0.5: BOOL;
	KU_VP1_out AT %QX8.30.0.6: BOOL;
	TZ_VP1_out AT %QX8.30.0.7: BOOL;

	input_Hz_LP4 AT %QW8.32.0: WORD; (*Задание входного значения часитоты*)
	input_Hz_LP5 AT %QW8.33.0: WORD; (*Задание входного значения часитоты*)
	LV_GR1_out AT %QW8.34.0: WORD;
	LV_LK7_out AT %QW8.35.0: WORD;
	LV_LK8_out AT %QW8.36.0: WORD;
	output_Hz_LP4_out AT %QW8.37.0: WORD;
	output_Hz_LP5_out AT %QW8.38.0: WORD;
	LV_D2_out AT %QW8.39.0: WORD;

	pusk_LAN_LP4 AT %QW8.48.0: WORD; (*Кнопка "пуск" из SCADA*)
	stop_LAN_LP4 AT %QW8.49.0: WORD; (*Кнопка "стоп" из SCADA*)
	pusk_LAN_LP5 AT %QW8.50.0: WORD; (*Кнопка "пуск" из SCADA*)
	stop_LAN_LP5 AT %QW8.51.0: WORD; (*Кнопка "стоп" из SCADA*)
	pusk_LAN_VP1 AT %QW8.52.0: WORD; (*Кнопка "пуск" из SCADA*)
	stop_LAN_VP1 AT %QW8.53.0: WORD; (*Кнопка "стоп" из SCADA*)
	pusk_lan_LK10 AT %QW8.54.0: WORD;
	pusk_lan_LK11 AT %QW8.55.0: WORD;

	pusk_lan_LK12 AT %QW8.56.0: WORD;
	pusk_lan_LK13 AT %QW8.57.0: WORD;
	pusk_lan_GR3 AT %QW8.58.0: WORD;
	pusk_lan_LK7 AT %QW8.59.0: WORD;
	pusk_lan_LK8 AT %QW8.60.0: WORD;
	pusk_lan_LK6 AT %QW8.61.0: WORD;
	pusk_lan_LK9 AT %QW8.62.0: WORD;
	pusk_lan_LP1_3 AT %QW8.63.0: WORD;

	pusk_lan_GR2 AT %QW8.64.0: WORD;
	pusk_lan_LK5 AT %QW8.65.0: WORD;
	pusk_lan_LK4 AT %QW8.66.0: WORD;
	pusk_lan_LK3 AT %QW8.67.0: WORD;
	pusk_lan_GR1 AT %QW8.68.0: WORD;
	pusk_lan_LK2 AT %QW8.69.0: WORD;
	stop_lan_LK10 AT %QW8.70.0: WORD;
	stop_lan_LK11 AT %QW8.71.0: WORD;

	stop_lan_LK12 AT %QW8.72.0: WORD;
	stop_lan_LK13 AT %QW8.73.0: WORD;
	stop_lan_GR3 AT %QW8.74.0: WORD;
	stop_lan_LK7 AT %QW8.75.0: WORD;
	stop_lan_LK8 AT %QW8.76.0: WORD;
	stop_lan_LK6 AT %QW8.77.0: WORD;
	stop_lan_LK9 AT %QW8.78.0: WORD;
	stop_lan_LP1_3 AT %QW8.79.0: WORD;

	stop_lan_GR2 AT %QW8.80.0: WORD;
	stop_lan_LK5 AT %QW8.81.0: WORD;
	stop_lan_LK4 AT %QW8.82.0: WORD;
	stop_lan_LK3 AT %QW8.83.0: WORD;
	stop_lan_GR1 AT %QW8.84.0: WORD;
	stop_lan_LK2 AT %QW8.85.0: WORD;

	stop_LAN_D3 AT %QW8.86.0: WORD;
	stop_LAN_D4 AT %QW8.87.0: WORD;

	stop_LAN_D2 AT %QW8.88.0: WORD;
	pusk_LAN_D2 AT %QW8.89.0: WORD;
	pusk_LAN_D3 AT %QW8.90.0: WORD;
	pusk_LAN_D4 AT %QW8.91.0: WORD;
	pusk_lan_cyclone AT %QW8.92.0: WORD;
	stop_lan_cyclone AT %QW8.93.0: WORD;
	revers AT %QW8.150.0: WORD; (*ручное управление реверсом, если не сработал датчик уровня*)

	avar_vl_lk10 AT %QX8.153.0.0: BOOL;
	avar_vl_lk11 AT %QX8.153.0.1: BOOL;
	avar_vl_lk12 AT %QX8.153.0.2: BOOL;
	avar_vl_lk13 AT %QX8.153.0.3: BOOL;
	avar_vl_lk7 AT %QX8.153.0.4: BOOL;
	avar_vl_lk8 AT %QX8.153.0.5: BOOL;
	avar_vl_lk6 AT %QX8.153.0.6: BOOL;
	avar_vl_lk9 AT %QX8.153.0.7: BOOL;

	avar_vl_lp1_3 AT %QX8.154.0.0: BOOL;
	avar_vl_lk5 AT %QX8.154.0.1: BOOL;
	avar_vl_lk4 AT %QX8.154.0.2: BOOL;
	avar_vl_lk3 AT %QX8.154.0.3: BOOL;
	avar_vl_lk2 AT %QX8.154.0.4: BOOL;
	avar_vl_lp4 AT %QX8.154.0.5: BOOL;
	avar_vl_lp5 AT %QX8.154.0.6: BOOL;
	gribok_out AT %QX8.154.0.7: BOOL;

	pusk_shnek_razg AT %QW8.155.0: WORD;
	stop_shnek_razg AT %QW8.156.0: WORD;

	TM_D3_word_out AT %QW8.157.0: WORD;
	TM_D4_word_out AT %QW8.158.0: WORD;

	avar_FC_LP4_out AT %QX8.159.0.0: BOOL;
	avar_FC_LP5_out AT %QX8.159.0.1: BOOL;
	e_lp4_temp_out AT %QX8.159.0.2: BOOL;
	e_d3_temp_out AT %QX8.159.0.3: BOOL;
	e_d4_temp_out AT %QX8.159.0.4: BOOL;
	e_vp1_temp_out AT %QX8.159.0.5: BOOL;
	lev_down_cyc_out AT %QX8.159.0.6: BOOL;
	moduls_out AT %QX8.159.0.7: BOOL;

	lk12_switcher AT %QW8.168.0: WORD;

	stop_vl_lv1: BOOL;
	stop_vl_lv2: BOOL;
	stop_vl_lv3: BOOL;

(*Блок сравнения введенных значений частот для ПЧ*)
	if_Hz: if_Hz;
	out_Hz_LP4: WORD;
	out_Hz_LP5: WORD;

(*Блок подачи разрешающего сигнала на ПП1*)
	PP1_blok: PP1;
	PP1 :BOOL (*коменда на отключение ПП1*);

(*Блок пробразования word-значений в bool-значегия для запуска агрегатов в ручном режиме*)
	signals1: bool_to;
	pusk_LAN_LP4_out: BOOL;
	stop_LAN_LP4_out: BOOL;
	pusk_LAN_LP5_out: BOOL;
	stop_LAN_LP5_out: BOOL;
	pusk_LAN_VP1_out: BOOL;
	stop_LAN_VP1_out: BOOL;
	pusk_lan_LK10_out: BOOL;
	pusk_lan_LK11_out: BOOL;
	pusk_lan_LK12_out: BOOL;
	pusk_lan_LK13_out: BOOL;
	pusk_lan_GR3_out: BOOL;
	pusk_lan_LK7_out: BOOL;
	pusk_lan_LK8_out: BOOL;
	pusk_lan_LK6_out: BOOL;
	pusk_lan_LK9_out: BOOL;
	pusk_lan_LP1_3_out: BOOL;
	pusk_lan_GR2_out: BOOL;
	pusk_lan_LK5_out: BOOL;
	pusk_lan_LK4_out: BOOL;
	pusk_lan_LK3_out: BOOL;
	pusk_lan_GR1_out: BOOL;
	pusk_lan_LK2_out: BOOL;
	stop_lan_LK10_out: BOOL;
	stop_lan_LK11_out: BOOL;
	stop_lan_LK12_out: BOOL;
	stop_lan_LK13_out: BOOL;
	stop_lan_GR3_out: BOOL;
	stop_lan_LK7_out: BOOL;
	stop_lan_LK8_out: BOOL;
	stop_lan_LK6_out: BOOL;
	stop_lan_LK9_out: BOOL;
	stop_lan_LP1_3_out: BOOL;
	stop_lan_GR2_out: BOOL;
	stop_lan_LK5_out: BOOL;
	stop_lan_LK4_out: BOOL;
	stop_lan_LK3_out: BOOL;
	stop_lan_GR1_out: BOOL;
	stop_lan_LK2_out: BOOL;
	pusk_LAN_D2_out: BOOL;
	stop_LAN_D2_out: BOOL;
	pusk_LAN_D3_out: BOOL;
	stop_LAN_D3_out: BOOL;
	stop_LAN_D4_out: BOOL;
	pusk_LAN_D4_out: BOOL;
	pusk_lan_cyclone_out: BOOL;
	stop_lan_cyclone_out: BOOL;

	tros_self_lk10_out: BOOL;
	shod_self_lk10_out: BOOL;
	ogr_self_lk10_out: BOOL;
	vl_self_lk10_out: BOOL;

	tros_self_lk11_out: BOOL;
	shod_self_lk11_out: BOOL;
	ogr_self_lk11_out: BOOL;
	vl_self_lk11_out: BOOL;

	tros_self_lk12_out: BOOL;
	shod_self_lk12_out: BOOL;
	ogr_self_lk12_out: BOOL;
	vl_self_lk12_out: BOOL;

	tros_self_lk13_out: BOOL;
	shod_self_lk13_out: BOOL;
	ogr_self_lk13_out: BOOL;
	vl_self_lk13_out: BOOL;

	tros_self_lk7_out: BOOL;
	shod_self_lk7_out: BOOL;
	ogr_self_lk7_out: BOOL;
	vl_self_lk7_out: BOOL;

	tros_self_lk8_out: BOOL;
	shod_self_lk8_out: BOOL;
	ogr_self_lk8_out: BOOL;
	vl_self_lk8_out: BOOL;

	tros_self_lk6_out: BOOL;
	shod_self_lk6_out: BOOL;
	ogr_self_lk6_out: BOOL;
	vl_self_lk6_out: BOOL;

	tros_self_lk9_out: BOOL;
	shod_self_lk9_out: BOOL;
	ogr_self_lk9_out: BOOL;
	vl_self_lk9_out: BOOL;
	vl_self_lp1_3_out: BOOL;

	tros_self_lk5_out: BOOL;
	shod_self_lk5_out: BOOL;
	ogr_self_lk5_out: BOOL;
	vl_self_lk5_out: BOOL;

	tros_self_lk4_out: BOOL;
	shod_self_lk4_out: BOOL;
	vl_self_lk4_out: BOOL;

	tros_self_lk3_out: BOOL;
	shod_self_lk3_out: BOOL;
	ogr_self_lk3_out: BOOL;
	vl_self_lk3_out: BOOL;

	tros_self_lk2_out: BOOL;
	shod_self_lk2_out: BOOL;
	ogr_self_lk2_out: BOOL;
	vl_self_lk2_out: BOOL;
	revers_out: BOOL;
	vl_self_lp4_out: BOOL;
	vl_self_lp5_out: BOOL;

	pusk_shnek_razg_out: BOOL;
	stop_shnek_razg_out: BOOL;

	prom10: BOOL;

	alarm_all: alarm_all;
	cyc_cleen_pusk: BOOL;
	cyc_cleen_stop: BOOL;

	prom_cleen_out AT %QW8.166.0: WORD;

	if_LV: if_LV;
END_VAR

VAR RETAIN PERSISTENT
	ust_LV2_GR1 AT %QD8.40.0: REAL;
	ust_LV1_GR1 AT %QD8.41.0: REAL;

	ust_LV2_LK7 AT %QD8.42.0: REAL;
	ust_LV1_LK7 AT %QD8.43.0: REAL;

	ust_LV2_LK8 AT %QD8.44.0: REAL;
	ust_LV1_LK8 AT %QD8.45.0: REAL;

	ust_LV2_D2 AT %QD8.46.0: REAL;
	ust_LV1_D2 AT %QD8.47.0: REAL;

	skvaj_in AT %QD8.94.0: REAL;

	tros_self_lk10 AT %QW8.102.0: WORD;
	shod_self_lk10 AT %QW8.103.0: WORD;
	ogr_self_lk10 AT %QW8.104.0: WORD;
	vl_self_lk10 AT %QW8.105.0: WORD;

	tros_self_lk11 AT %QW8.106.0: WORD;
	shod_self_lk11 AT %QW8.107.0: WORD;
	ogr_self_lk11 AT %QW8.108.0: WORD;
	vl_self_lk11 AT %QW8.109.0: WORD;

	tros_self_lk12 AT %QW8.110.0: WORD;
	shod_self_lk12 AT %QW8.111.0: WORD;
	ogr_self_lk12 AT %QW8.112.0: WORD;
	vl_self_lk12 AT %QW8.113.0: WORD;

	tros_self_lk13 AT %QW8.114.0: WORD;
	shod_self_lk13 AT %QW8.115.0: WORD;
	ogr_self_lk13 AT %QW8.116.0: WORD;
	vl_self_lk13 AT %QW8.117.0: WORD;

	tros_self_lk7 AT %QW8.118.0: WORD;
	shod_self_lk7 AT %QW8.119.0: WORD;
	ogr_self_lk7 AT %QW8.120.0: WORD;
	vl_self_lk7 AT %QW8.121.0: WORD;

	tros_self_lk8 AT %QW8.122.0: WORD;
	shod_self_lk8 AT %QW8.123.0: WORD;
	ogr_self_lk8 AT %QW8.124.0: WORD;
	vl_self_lk8 AT %QW8.125.0: WORD;

	tros_self_lk6 AT %QW8.126.0: WORD;
	shod_self_lk6 AT %QW8.127.0: WORD;
	ogr_self_lk6 AT %QW8.128.0: WORD;
	vl_self_lk6 AT %QW8.129.0: WORD;

	tros_self_lk9 AT %QW8.130.0: WORD;
	shod_self_lk9 AT %QW8.131.0: WORD;
	ogr_self_lk9 AT %QW8.132.0: WORD;
	vl_self_lk9 AT %QW8.133.0: WORD;
	vl_self_lp1_3 AT %QW8.134.0: WORD;

	tros_self_lk5 AT %QW8.135.0: WORD;
	shod_self_lk5 AT %QW8.136.0: WORD;
	ogr_self_lk5 AT %QW8.137.0: WORD;
	vl_self_lk5 AT %QW8.138.0: WORD;

	tros_self_lk4 AT %QW8.139.0: WORD;
	shod_self_lk4 AT %QW8.140.0: WORD;
	vl_self_lk4 AT %QW8.141.0: WORD;

	tros_self_lk3 AT %QW8.142.0: WORD;
	shod_self_lk3 AT %QW8.143.0: WORD;
	ogr_self_lk3 AT %QW8.144.0: WORD;
	vl_self_lk3 AT %QW8.145.0: WORD;

	tros_self_lk2 AT %QW8.146.0: WORD;
	shod_self_lk2 AT %QW8.147.0: WORD;
	ogr_self_lk2 AT %QW8.148.0: WORD;
	vl_self_lk2 AT %QW8.149.0: WORD;

	vl_self_lp4 AT %QW8.151.0: WORD;
	vl_self_lp5 AT %QW8.152.0: WORD;

	in_time_shake AT %QW8.160.0: WORD; (*пауза между встряхиваниями*)
	time_VL AT %QW8.161.0: WORD; (*задержка на отключение конвееров по скорости*)

	time_run AT %QW8.162.0: WORD; (*время работы *)
	time_stop AT %QW8.163.0: WORD; (*задержка на отключение конвееров по скорости*)

	pusk_cleen_lan AT %QW8.164.0: WORD;
	stop_cleen_lan AT %QW8.165.0: WORD;

	current_value_lk_glob AT %QX8.29.0.6: BOOL;
END_VAR
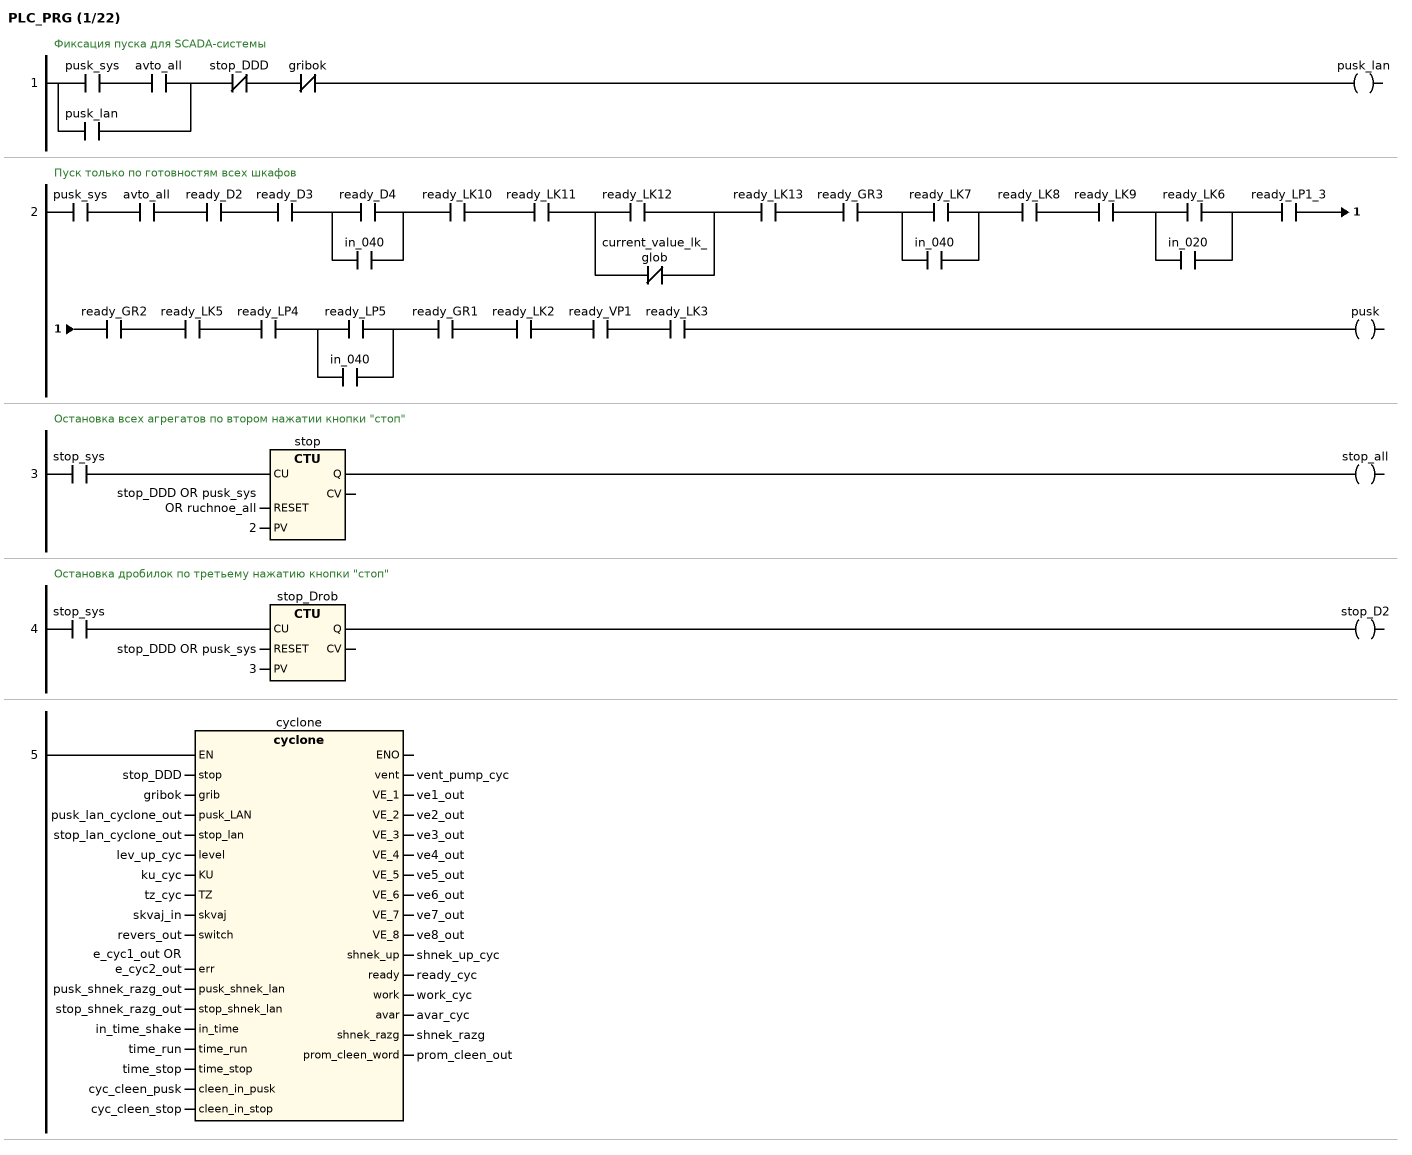
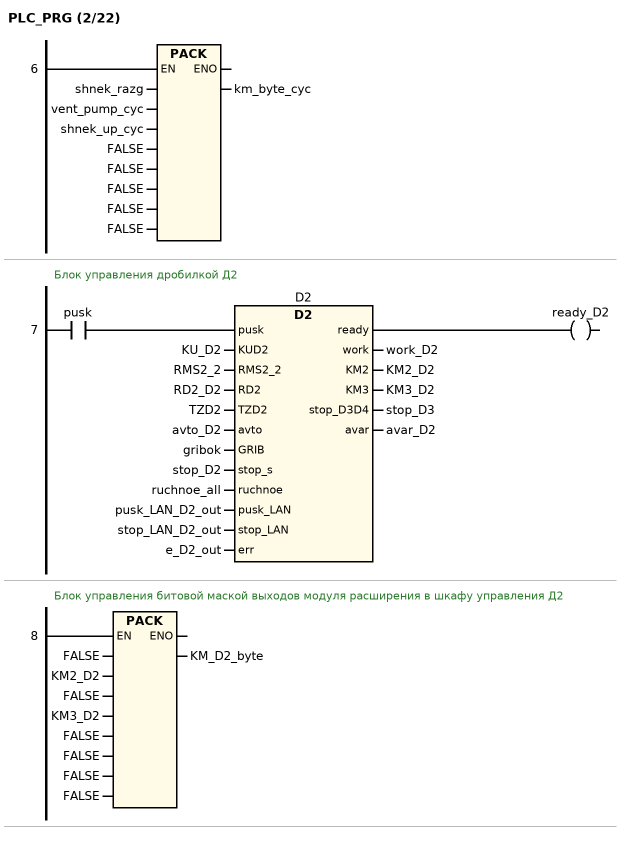
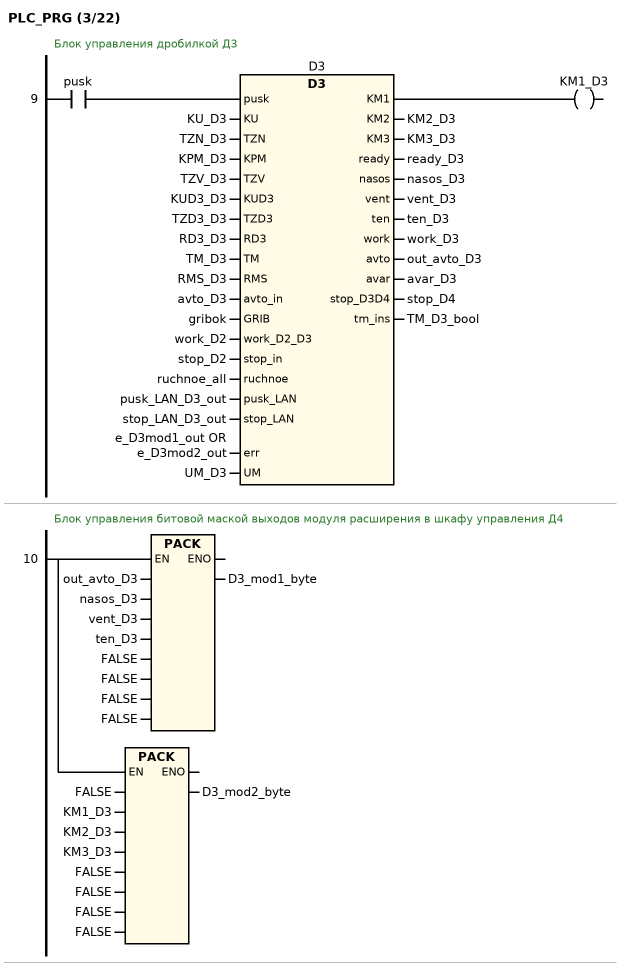
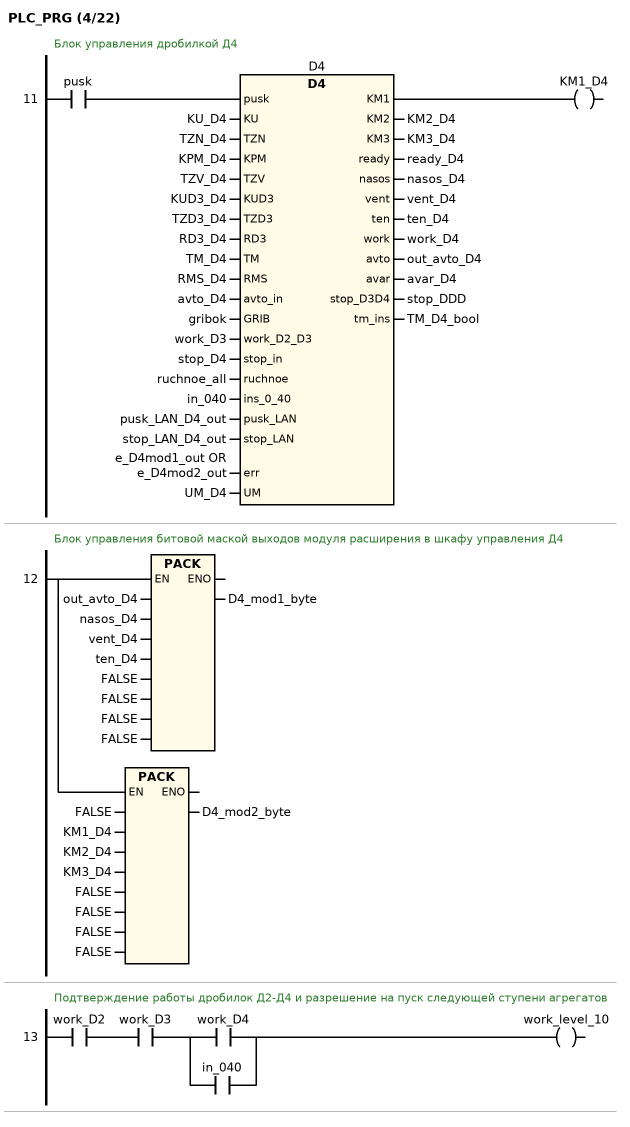
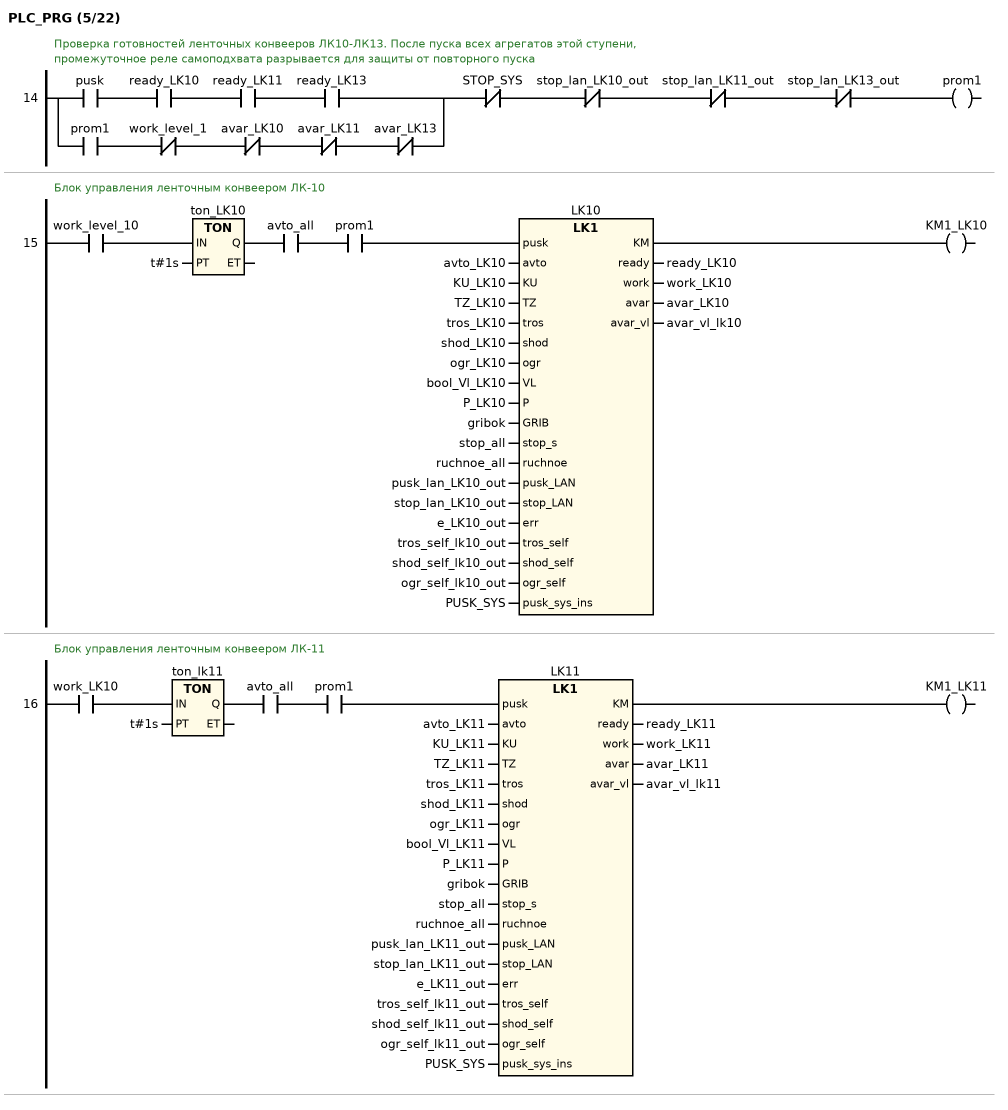
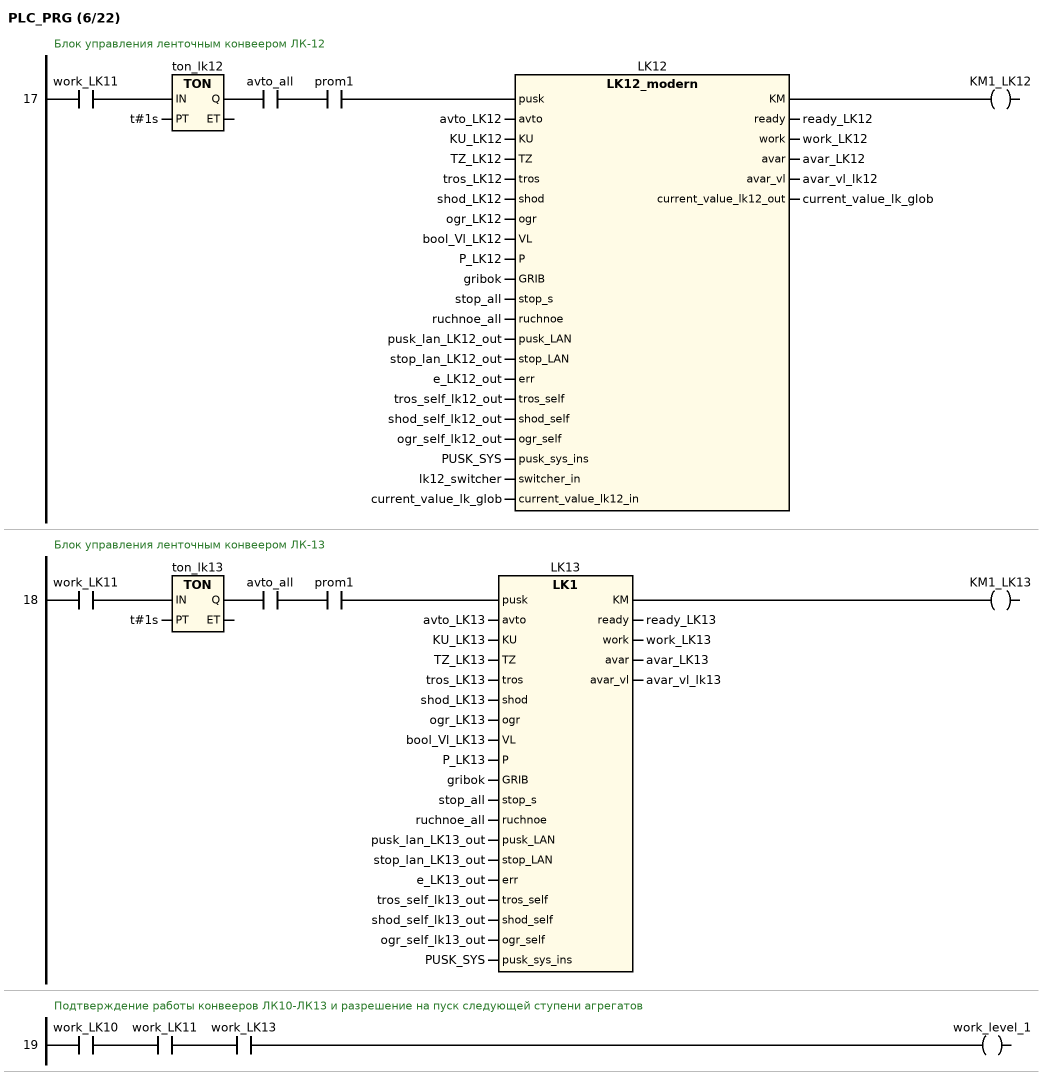
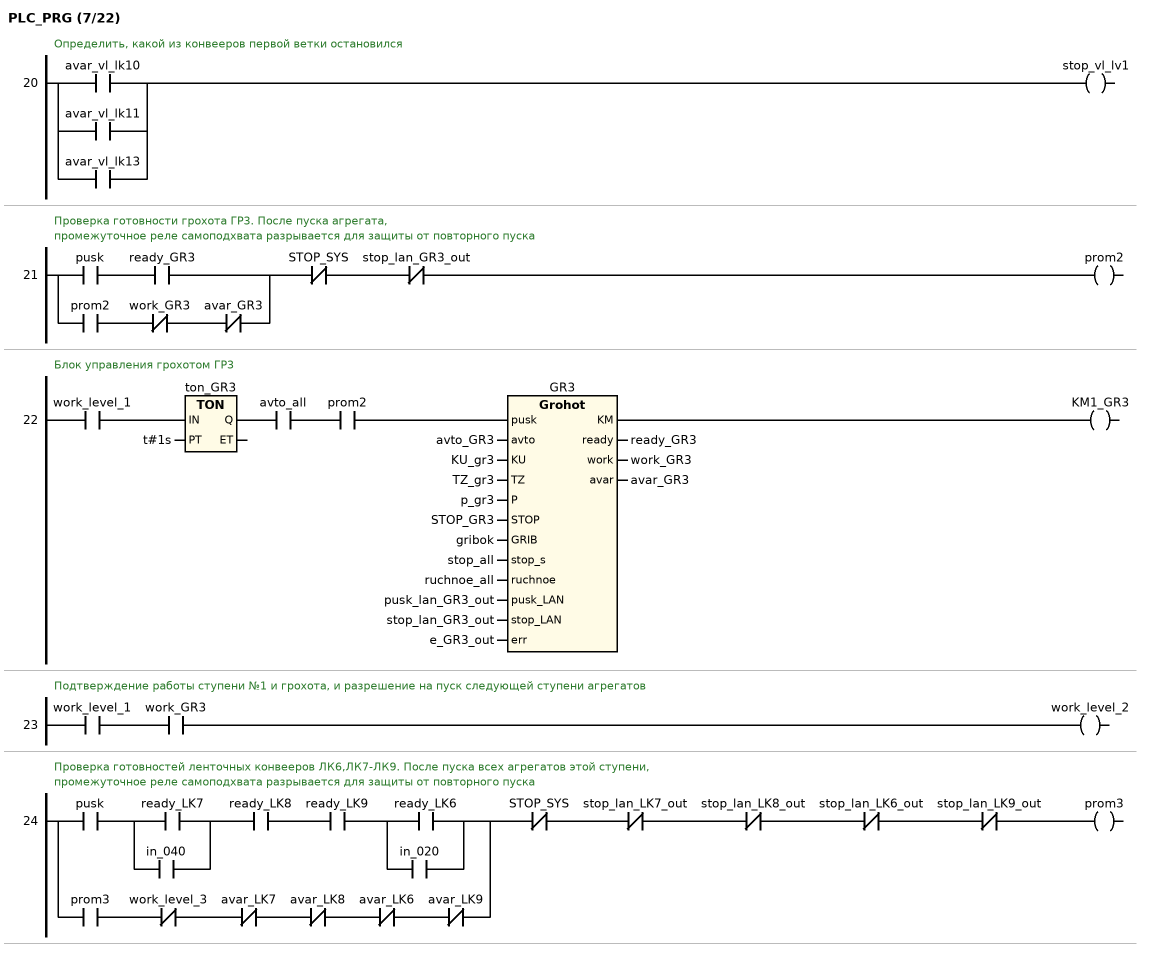
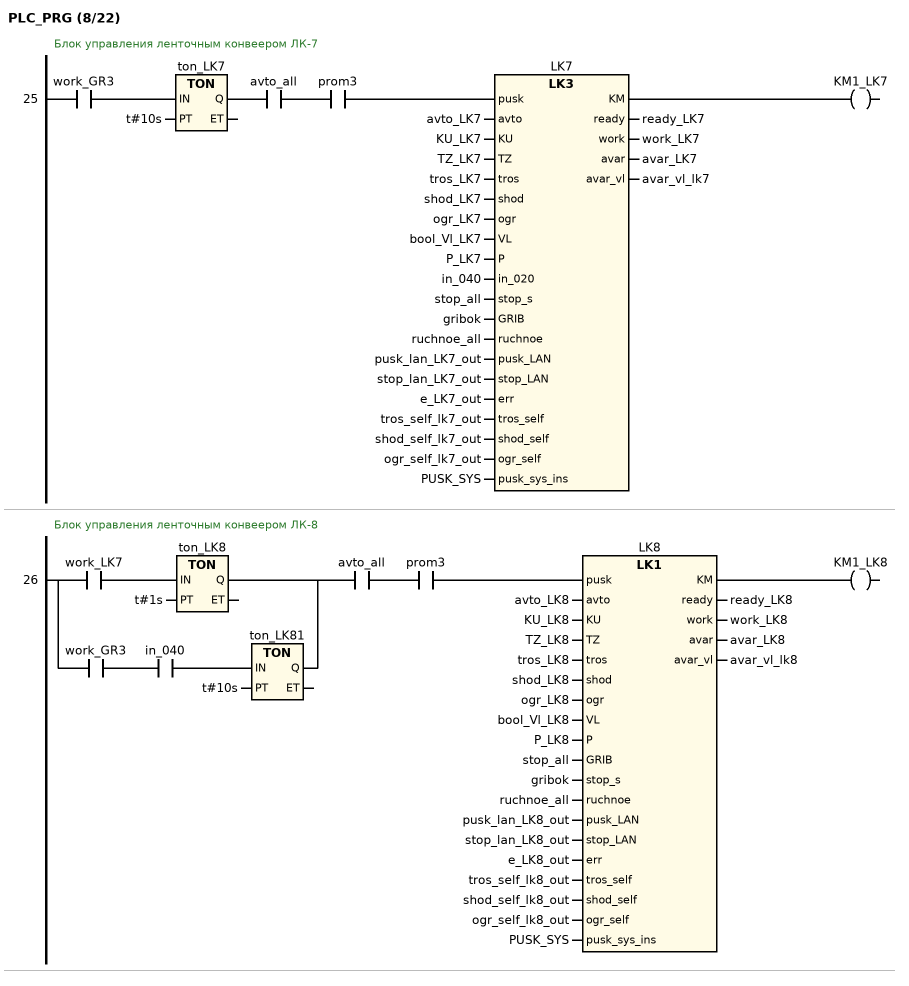
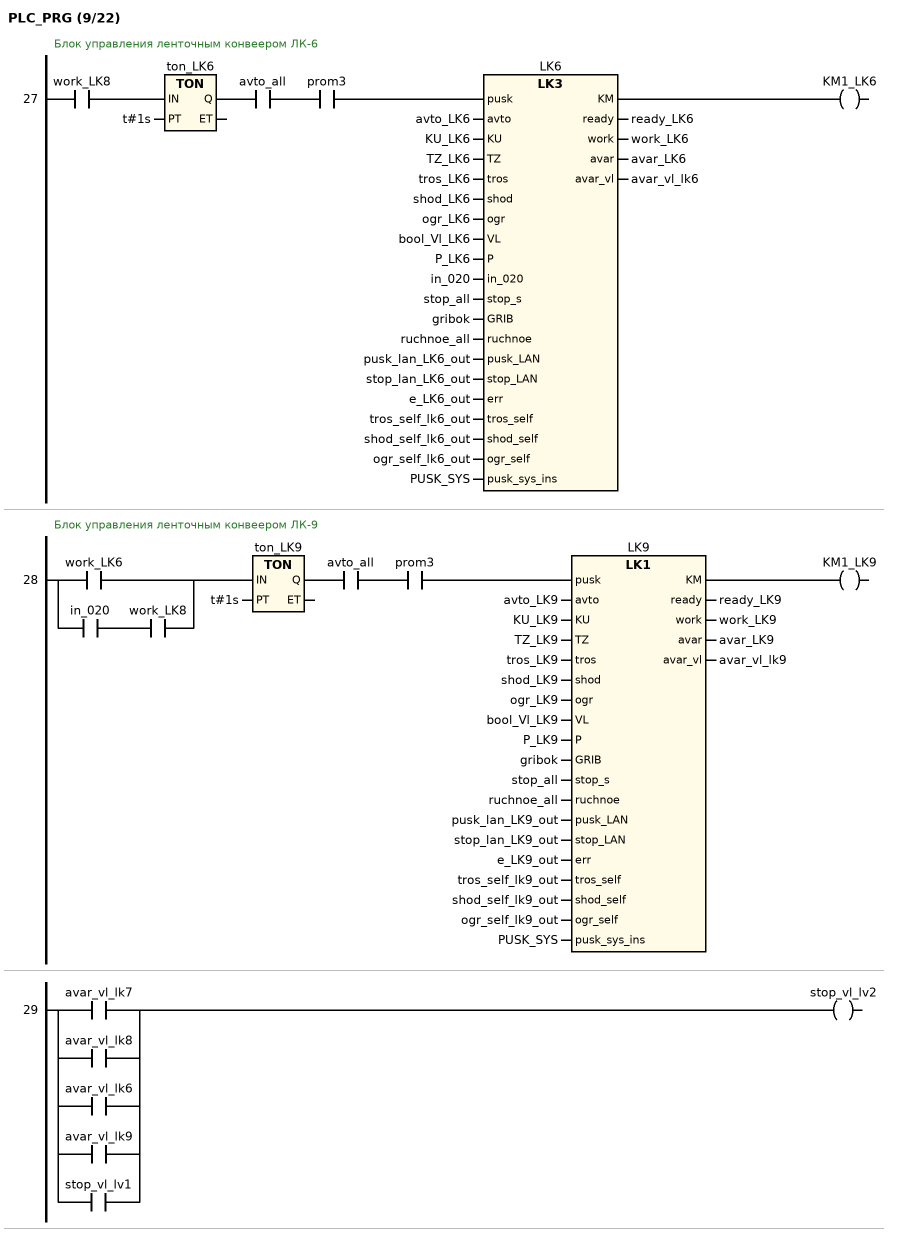
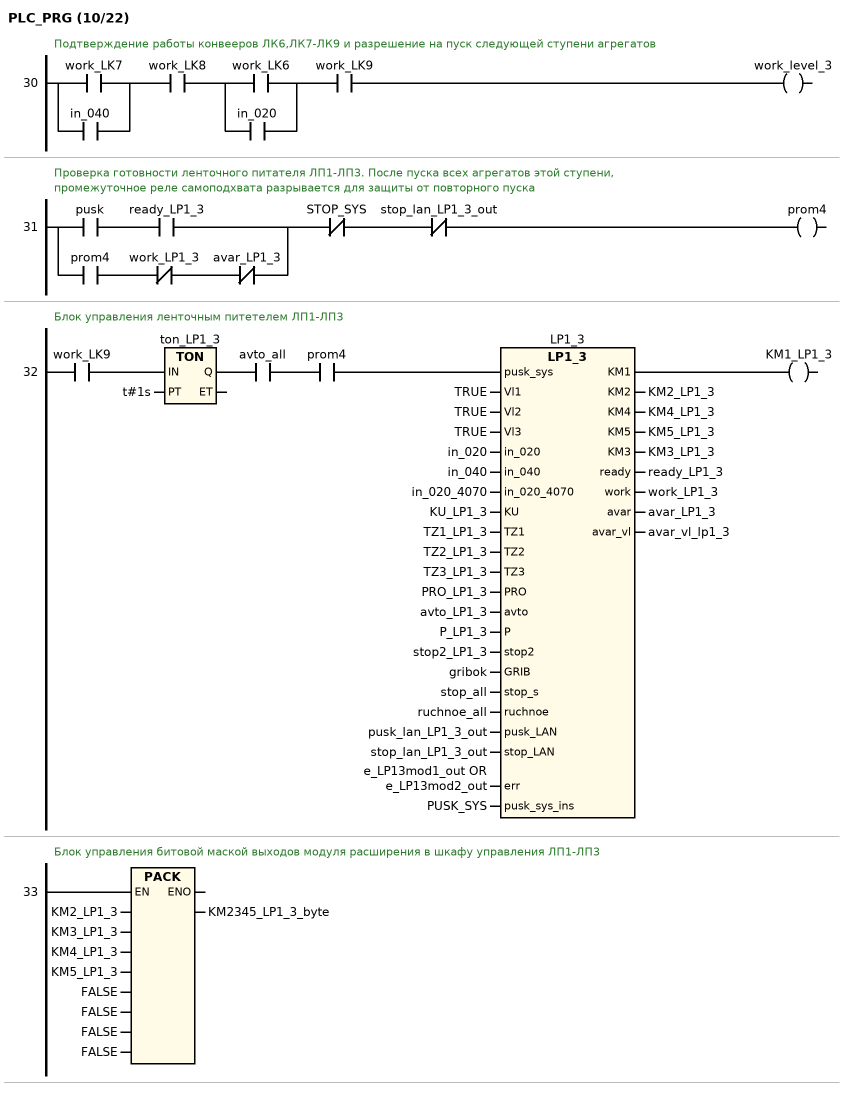
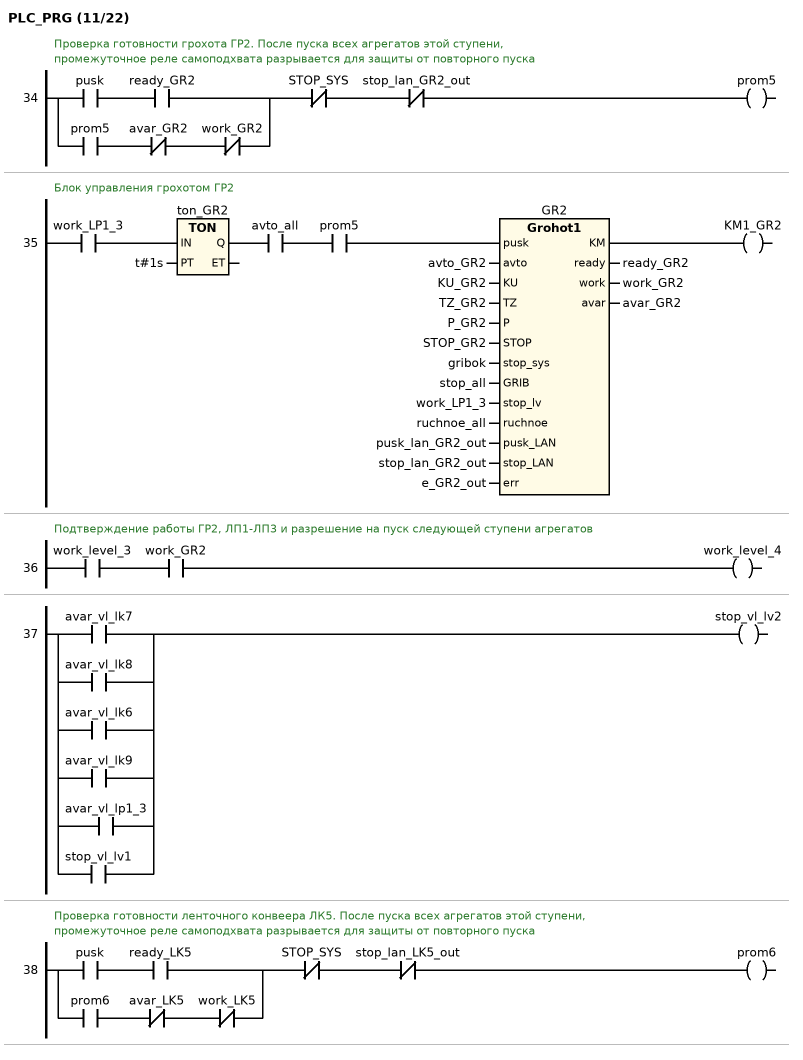
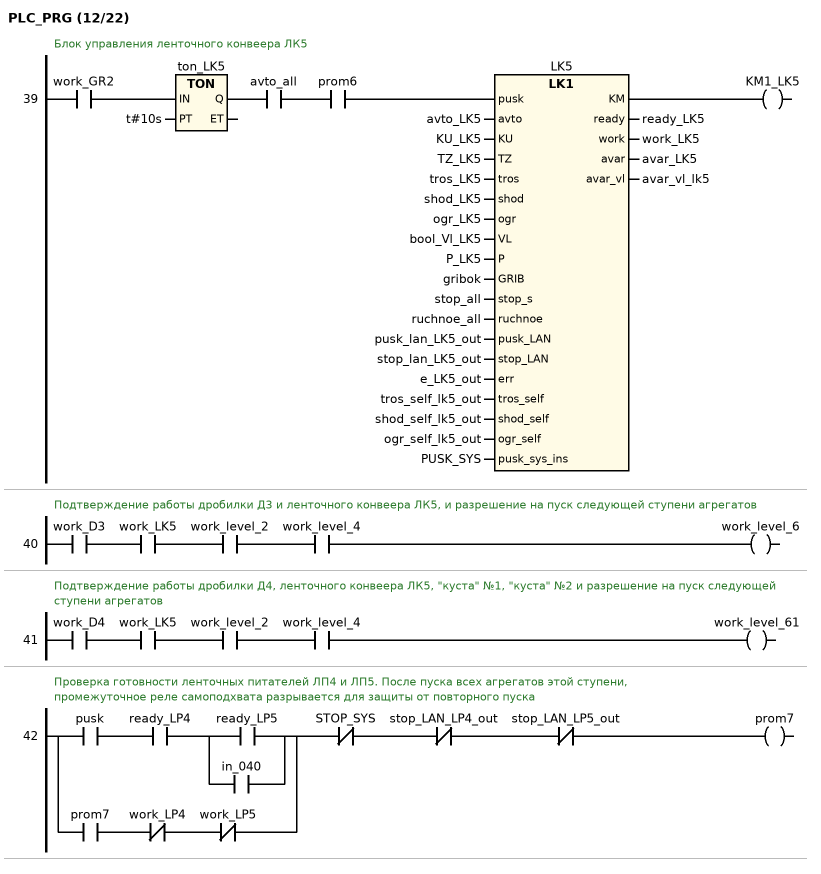
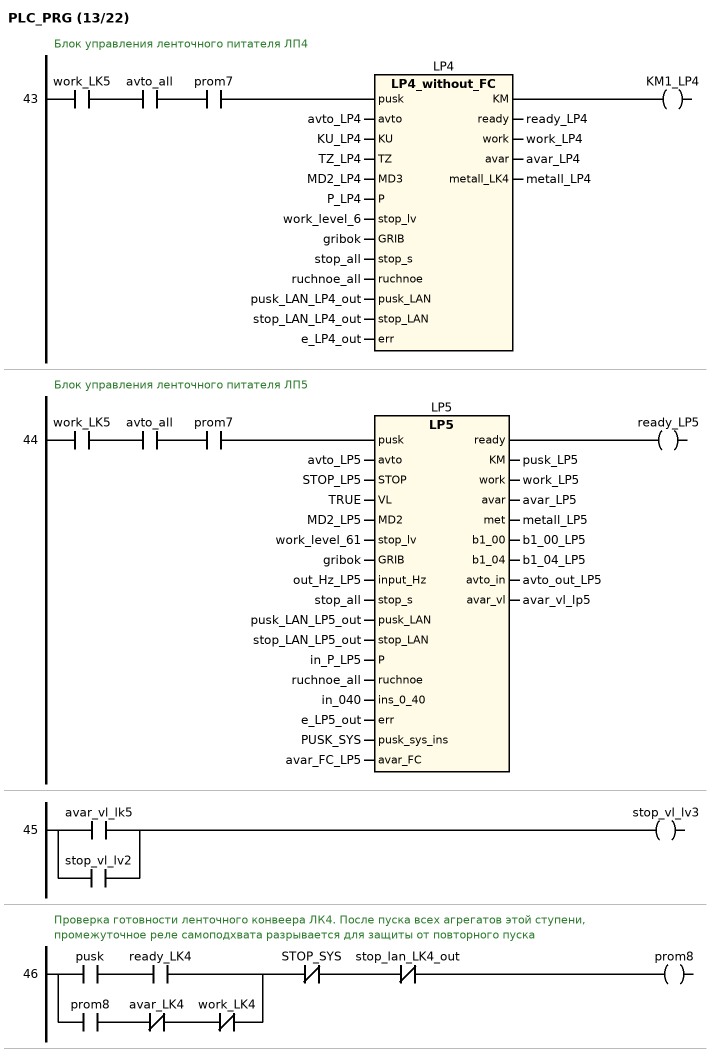
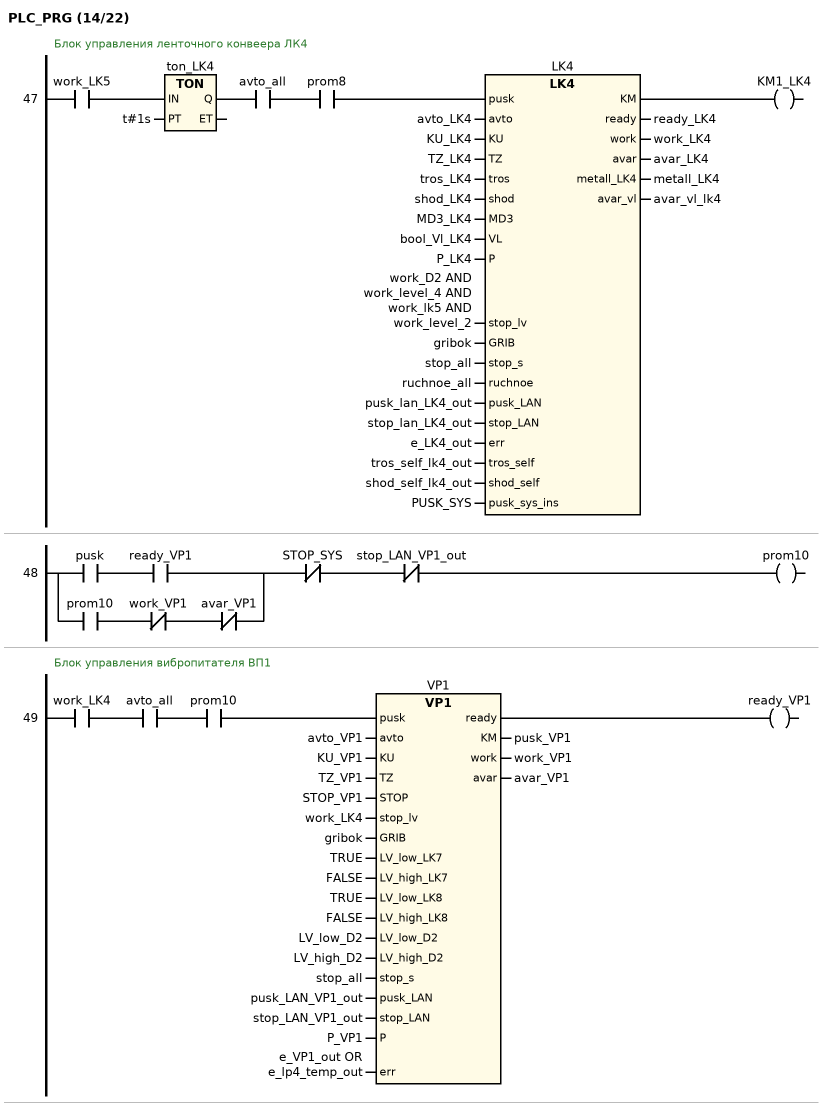
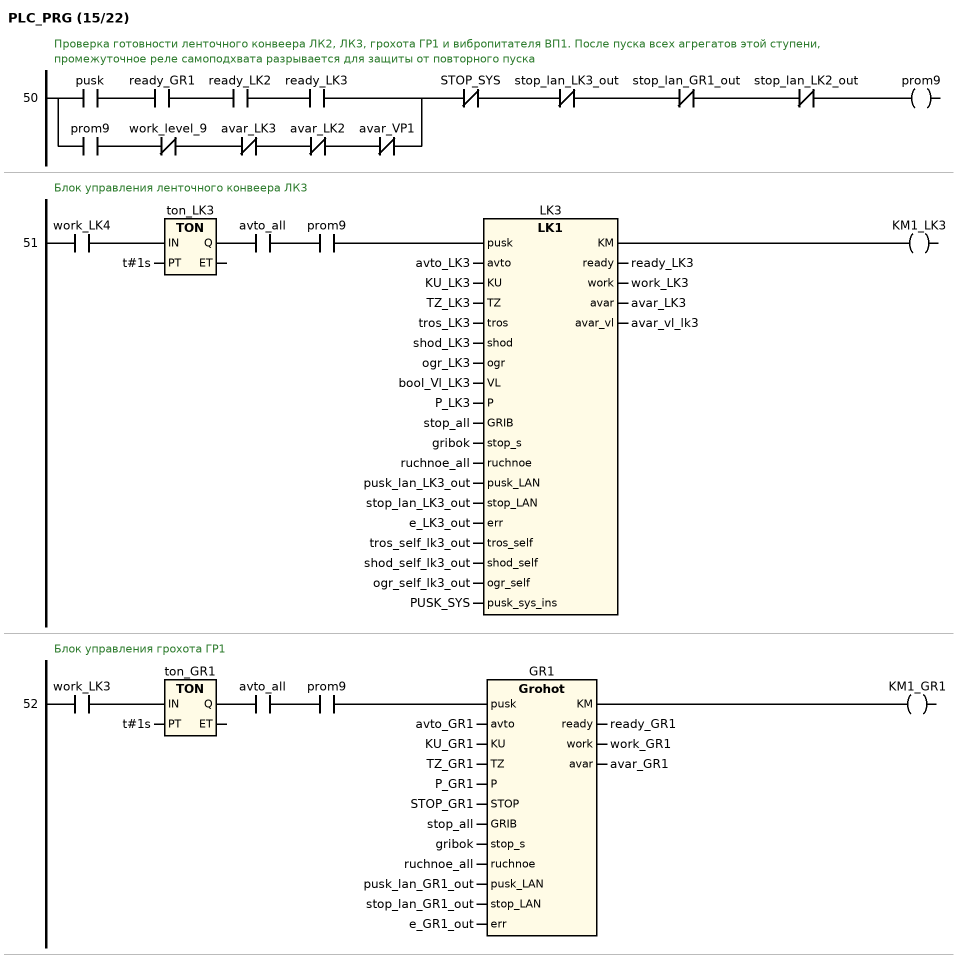
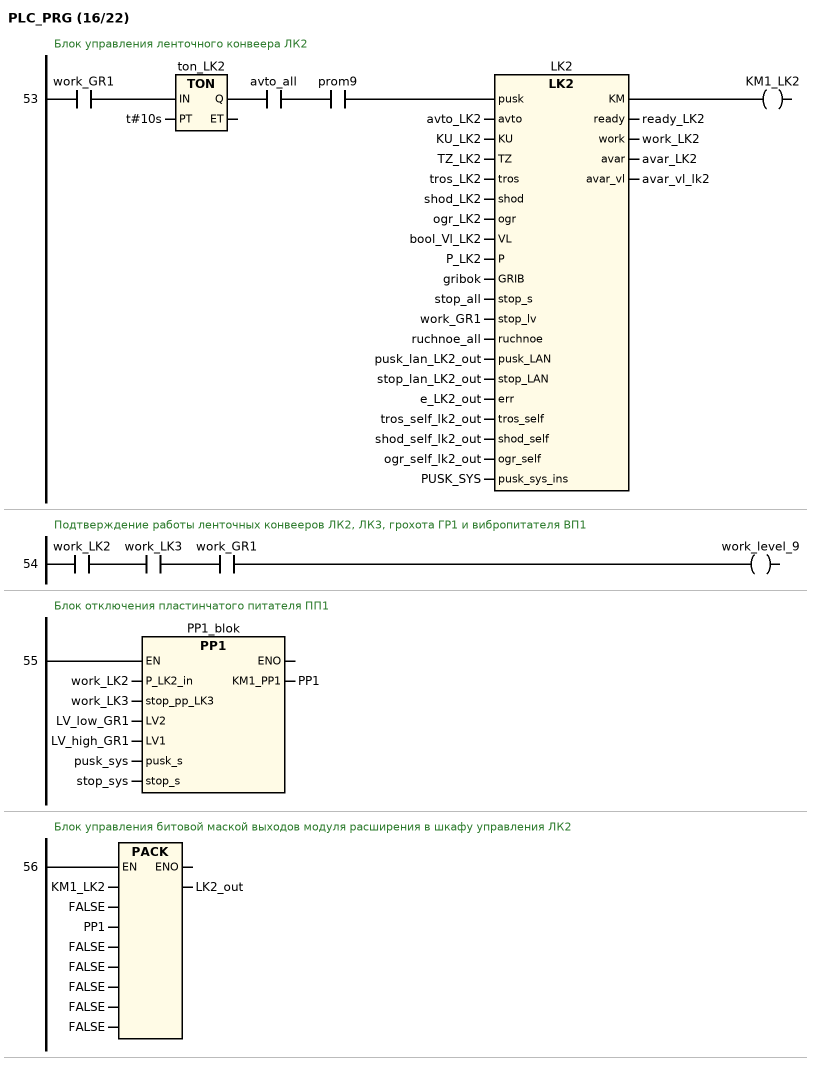
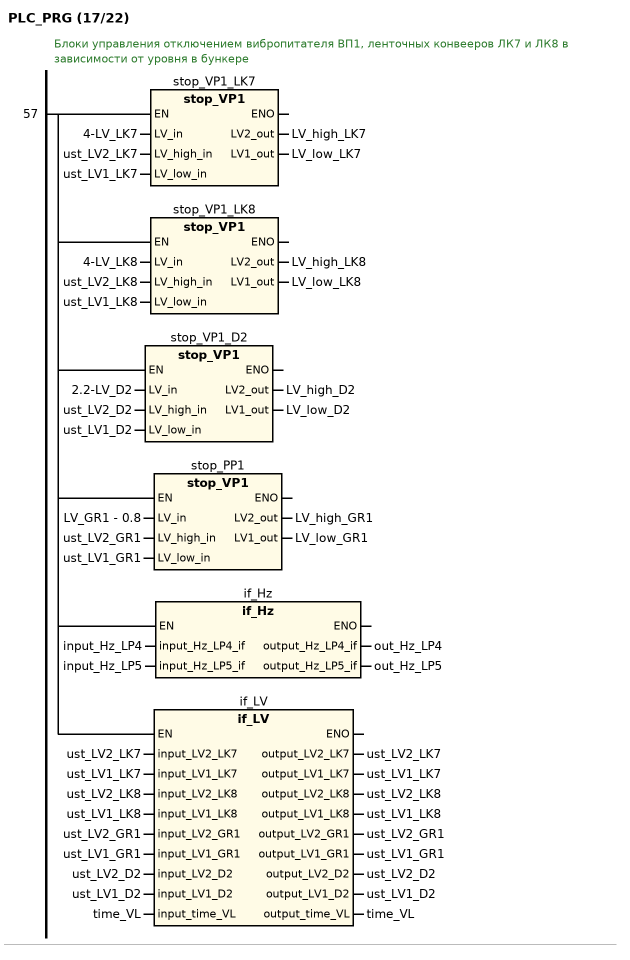
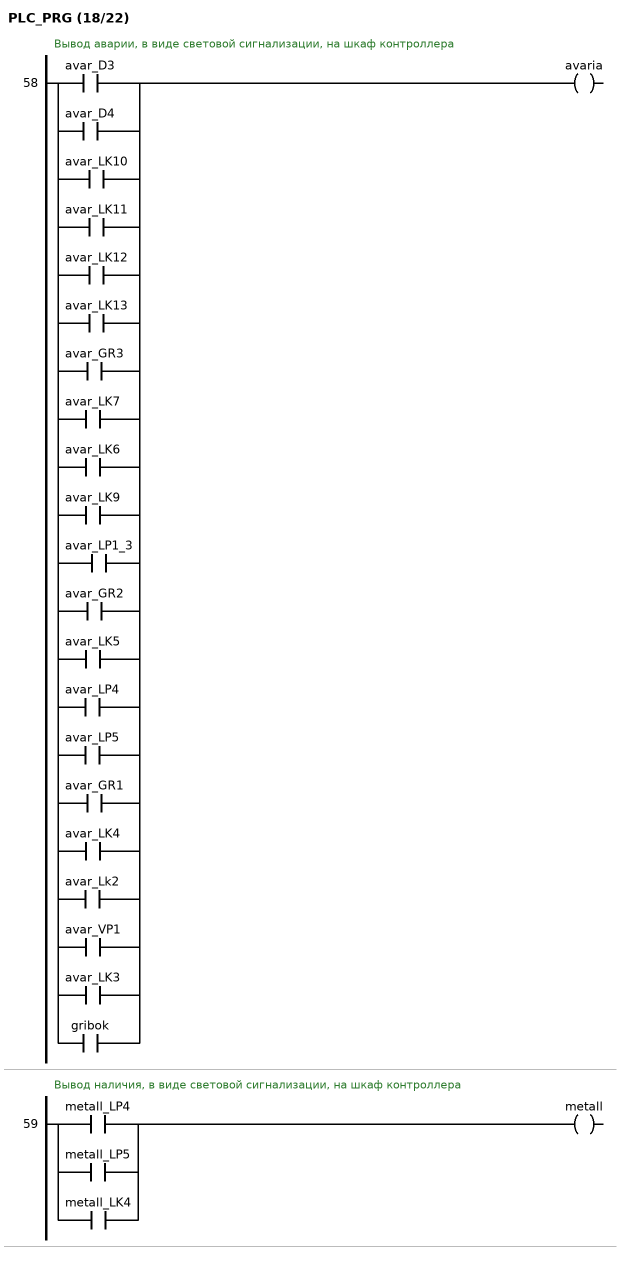
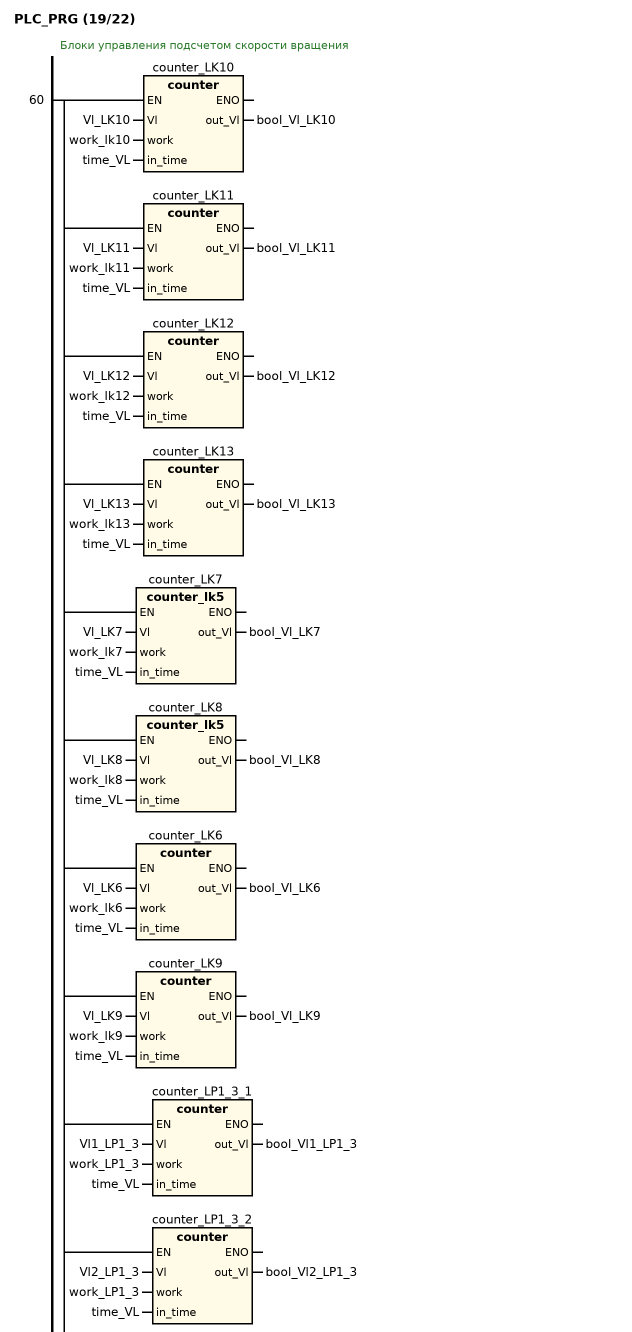
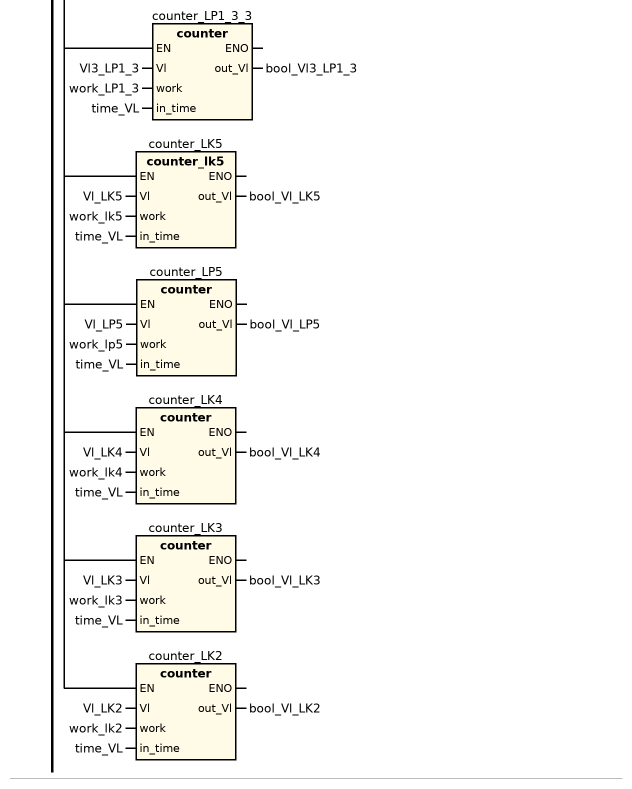
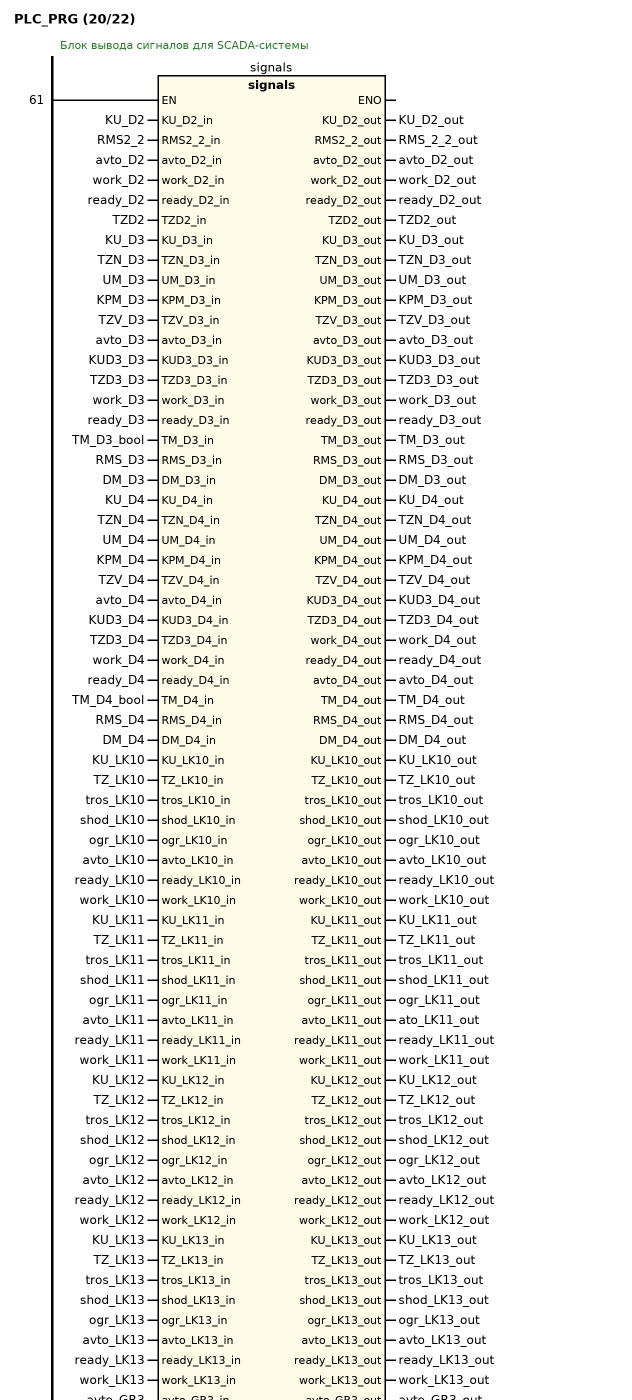
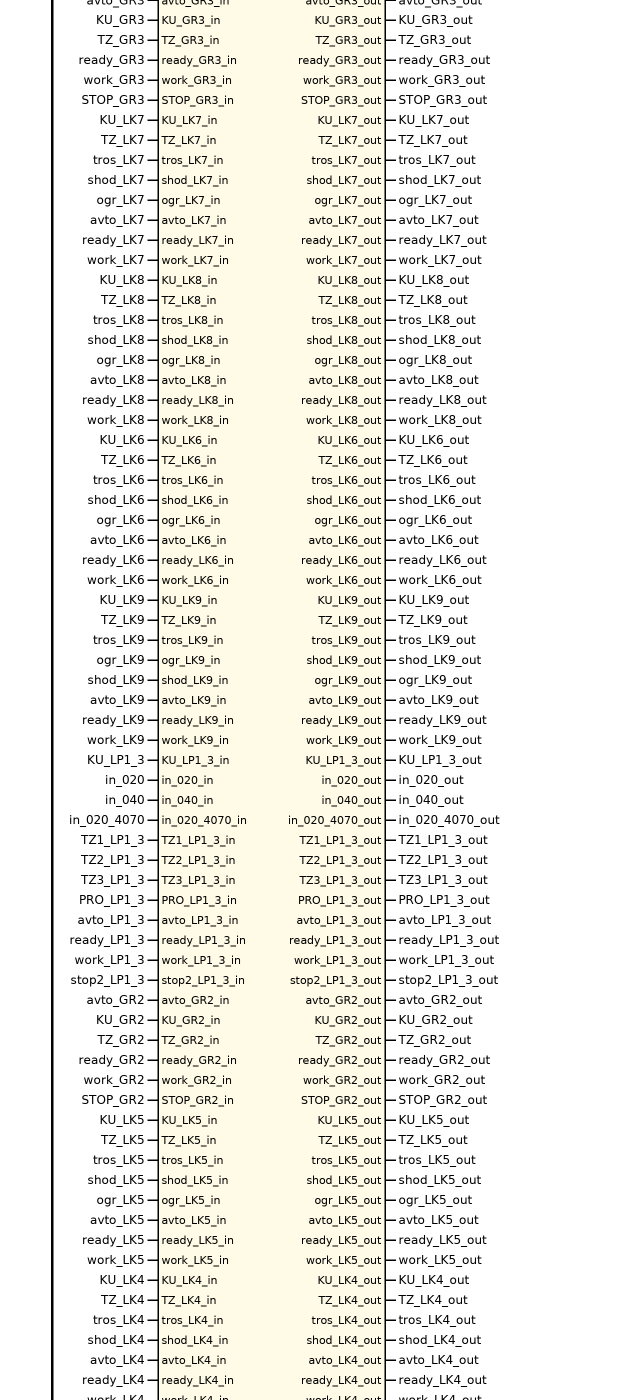
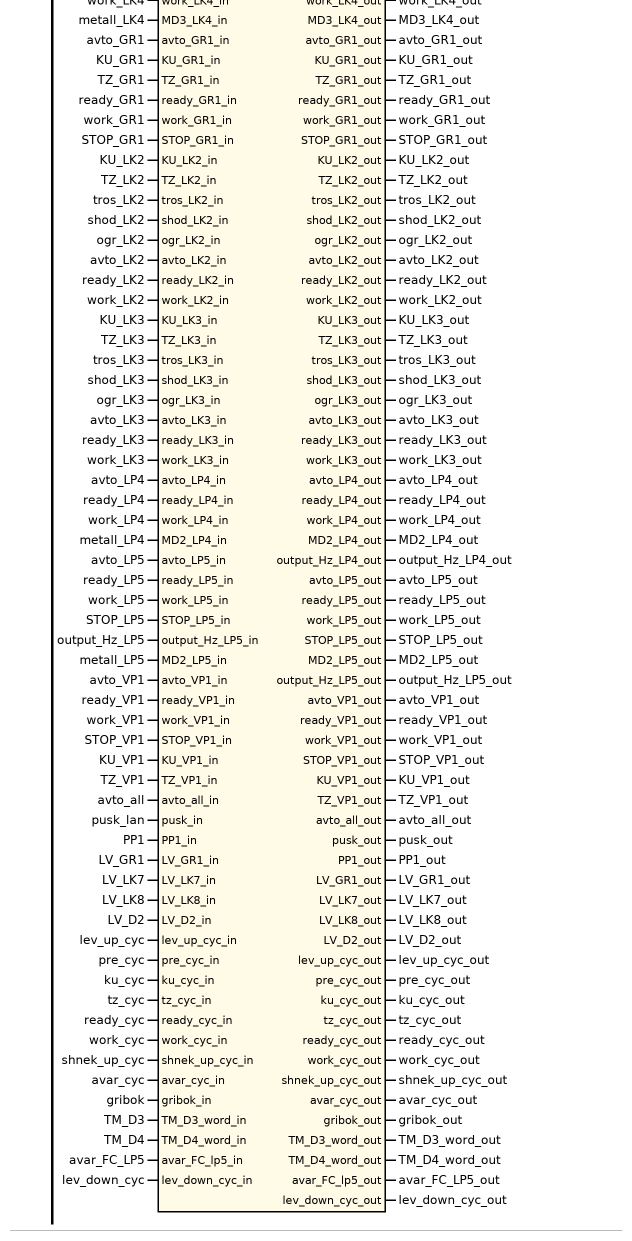
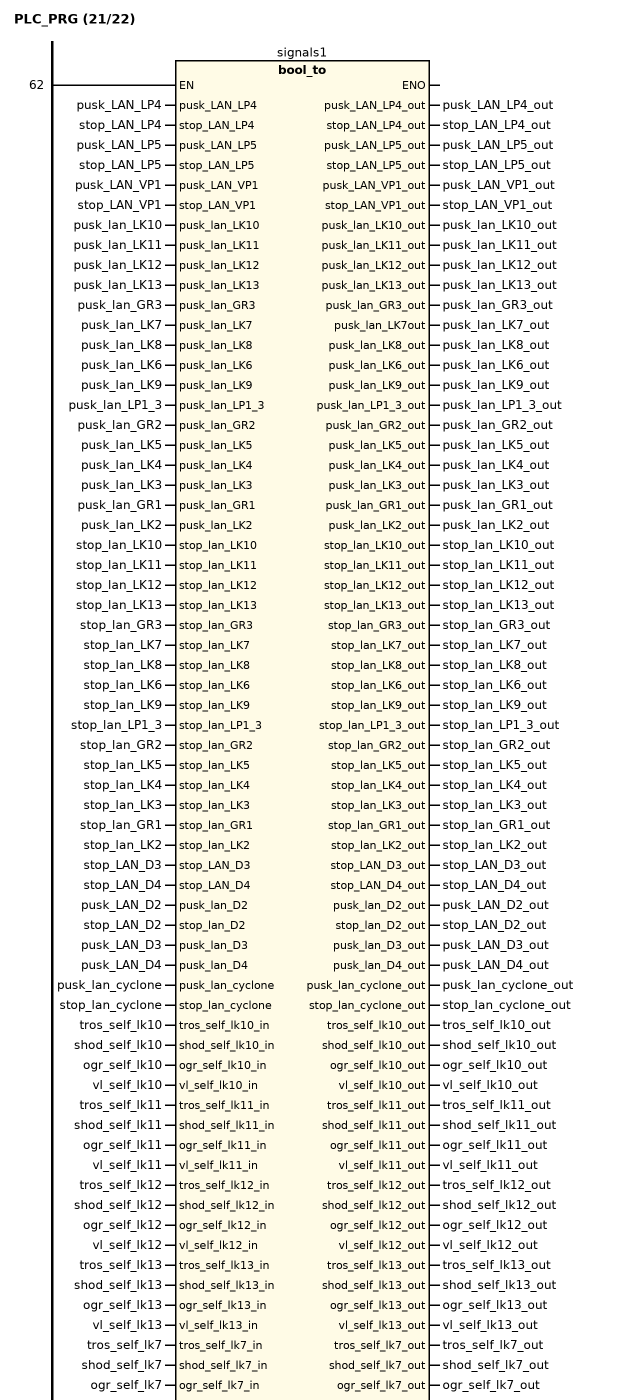
